// TwinCAT 3 PLC project PLC_1
// ProgramVersion: 3.1.4020.4
// libraries:
//   Tc2_ModbusSrv, * (Beckhoff Automation GmbH)
//   Tc2_Standard, * (Beckhoff Automation GmbH)
//   Tc2_System, * (Beckhoff Automation GmbH)
//   Tc2_TcpIp, * (Beckhoff Automation GmbH)
//   Tc2_Utilities, * (Beckhoff Automation GmbH)
//   Tc3_Module, * (Beckhoff Automation GmbH)
//   VisuDialogs, * (System)
// project tree:
//   DUTs/ E_RobotTaskStates.TcDUT, E_ProcessModes.TcDUT, E_RobotDataRecordingStates.TcDUT, E_UDPConnection.TcDUT, ST_16Bool.TcDUT, ST_Fixture.TcDUT, ST_OptoforceUDPData.TcDUT, ST_OptoforceUDPRequest.TcDUT, ST_Part.TcDUT, ST_RobotTaskStatusInfo.TcDUT, ST_UR.TcDUT
//   DUTs/UR_TCP_IP_Data_Collection_DUTs/ E_RobotTCPReceive.TcDUT, ST_AdditionalInfo.TcDUT, ST_CalibraitonData.TcDUT, ST_CartesianInfo.TcDUT, ST_ConfigurationData.TcDUT, ST_ForceModeData.TcDUT, ST_JointData.TcDUT, ST_KinematicInfo.TcDUT, ST_MasterboardData.TcDUT, ST_PackageInfo.TcDUT, ST_RobotModeData.TcDUT, ST_ToolData.TcDUT
//   / GlobalTextList.TcGTLO, PlcTask.TcTTO, Visualization Manager.TcVMO (not stored)
//   GVLs/ Global.TcGVL, Global_Safety.TcGVL
//   POUs/ FB_CSV_PartDataWriter.TcPOU, FB_CSV_RobotDataWriter.TcPOU, FB_CSV_FTDataWriter.TcPOU, FB_FT_UDPConnection.TcPOU, MAIN.TcPOU, F_Word_To_16Bool.TcPOU, P_InitializeSystem.TcPOU, P_InputOutputHandling.TcPOU, P_Safety.TcPOU, P_TaskHandling.TcPOU
//   POUs/Modbus POUs/ FB_mbReadSingleReg.TcPOU, FB_mbReadRobotTaskStatusInfo.TcPOU, FB_mbWriteRobotTask.TcPOU, FB_mbWriteSingleReg.TcPOU
//   POUs/UR_TCP_IP_Data_Collection/ FB_ParseURData.TcPOU, FB_RobotTCPReceive.TcPOU, F_RecCartesianInfo.TcPOU, F_RecJointData.TcPOU, F_RecRobotModeData.TcPOU, F_RecConfigurationData.TcPOU, F_FindAddr.TcPOU, F_RecForceModeData.TcPOU
//   VISUs/ ForceAndTorque.TcVIS, PositionCheck.TcVIS, Settings.TcVIS, Process.TcVIS, TopVisu.TcVIS
// real-time tasks:
//   TASK PlcTask: cycle T#1ms, priority 20, ADS port 350
// I/O:
//   DEVICE Device 1 (EtherCAT), AmsNetId 5.43.59.116.2.1
//     Term 1 (EK1200) [EK1200-5000 EtherCAT Power supply (2A E-Bus)]
//       SafetyPLC (EL6900) [EL6900, TwinSAFE PLC]
//       Safe In - E-Stop & Reset (EL1904) [EL1904, 4 Ch. Safety Input 24V, TwinSAFE]
//         modules: Module 1 (FSOES)
//       Safe In - Programming Mode (EL1904) [EL1904, 4 Ch. Safety Input 24V, TwinSAFE]
//         modules: Module 1 (FSOES)
//       In - Control Buttons (EL1014) [EL1014 4Ch. Dig. Input 24V, 10µs]
//       In - Unused (EL1014) [EL1014 4Ch. Dig. Input 24V, 10µs]
//       Out - Control Button Ind. (EL2004) [EL2004 4Ch. Dig. Output 24V, 0.5A]
//       Out - Prog. Mode Ind. (EL2004) [EL2004 4Ch. Dig. Output 24V, 0.5A]
//       EtherCAT Extender (EK1110) [EK1110 EtherCAT extension]
//     Term 10 (EK1100) [EK1100 EtherCAT Coupler (2A E-Bus)]
//       In 2/3 wire - Unused 1 (EL1012) [EL1012 2Ch. Dig. Input 24V, 10µs]
//       Safe In - Robot E-Stop Cond. (EL1904) [EL1904, 4 Ch. Safety Input 24V, TwinSAFE]
//         modules: Module 1 (FSOES)
//       Safe In - E-Stop and Mats (EL1904) [EL1904, 4 Ch. Safety Input 24V, TwinSAFE]
//         modules: Module 1 (FSOES)
//       Safe In - Safety Laser A (horizontal) (EL1904) [EL1904, 4 Ch. Safety Input 24V, TwinSAFE]
//         modules: Module 1 (FSOES)
//       Safe In - Safety Laser B (vertical)  (EL1904) [EL1904, 4 Ch. Safety Input 24V, TwinSAFE]
//         modules: Module 1 (FSOES)
//       Safe Out - Robot Safety States (EL2904) [EL2904, 4 Ch. Safety Output 24V, 0.5A, TwinSAFE]
//         modules: Module 1 (FSOES), Module 2 (DO)
//       Out - Stack Lights (EL2008) [EL2008 8Ch. Dig. Output 24V, 0.5A]
//       In - General 1-wire (EL1018) [EL1018 8Ch. Dig. Input 24V, 10µs]
//       In - Unused 3 (EL1114) [EL1114 4Ch. Dig. Input 24V, 10µs, Sensor Power]
//       End Cap (passive) (EL9011) [EL9011 End Terminal]
// variable links:
//   Device 1 (EtherCAT) <-> Device 1 (EtherCAT)/Term 1 (EK1200)/SafetyPLC (EL6900)
//     Term 1 (EK1200)/Safe In - E-Stop & Reset (EL1904)/Module 1 (FSOES)/RxPDO/FSOE <-> ConnectionInputs/Message_3 TxPDO
//     Term 1 (EK1200)/Safe In - E-Stop & Reset (EL1904)/Module 1 (FSOES)/TxPDO/FSOE <-> ConnectionOutputs/Message_3 RxPDO
//     Term 1 (EK1200)/Safe In - Programming Mode (EL1904)/Module 1 (FSOES)/RxPDO/FSOE <-> ConnectionInputs/Message_15 TxPDO
//     Term 1 (EK1200)/Safe In - Programming Mode (EL1904)/Module 1 (FSOES)/TxPDO/FSOE <-> ConnectionOutputs/Message_15 RxPDO
//     Term 10 (EK1100)/Safe In - E-Stop and Mats (EL1904)/Module 1 (FSOES)/RxPDO/FSOE <-> ConnectionInputs/Message_6 TxPDO
//     Term 10 (EK1100)/Safe In - E-Stop and Mats (EL1904)/Module 1 (FSOES)/TxPDO/FSOE <-> ConnectionOutputs/Message_6 RxPDO
//     Term 10 (EK1100)/Safe In - Robot E-Stop Cond. (EL1904)/Module 1 (FSOES)/RxPDO/FSOE <-> ConnectionInputs/Message_14 TxPDO
//     Term 10 (EK1100)/Safe In - Safety Laser A (horizontal) (EL1904)/Module 1 (FSOES)/RxPDO/FSOE <-> ConnectionInputs/Message_16 TxPDO
//     Term 10 (EK1100)/Safe In - Safety Laser A (horizontal) (EL1904)/Module 1 (FSOES)/TxPDO/FSOE <-> ConnectionOutputs/Message_16 RxPDO
//     Term 10 (EK1100)/Safe In - Safety Laser B (vertical)  (EL1904)/Module 1 (FSOES)/RxPDO/FSOE <-> ConnectionInputs/Message_18 TxPDO
//     Term 10 (EK1100)/Safe Out - Robot Safety States (EL2904)/Module 1 (FSOES)/RxPDO/FSOE <-> ConnectionInputs/Message_9 TxPDO
//   Device 1 (EtherCAT) <-> Device 1 (EtherCAT)/Term 10 (EK1100)/Safe In - Robot E-Stop Cond. (EL1904)
//     Term 1 (EK1200)/SafetyPLC (EL6900)/ConnectionOutputs/Message_14 RxPDO <-> Module 1 (FSOES)/TxPDO/FSOE
//   Device 1 (EtherCAT) <-> Device 1 (EtherCAT)/Term 10 (EK1100)/Safe In - Safety Laser B (vertical)  (EL1904)
//     Term 1 (EK1200)/SafetyPLC (EL6900)/ConnectionOutputs/Message_18 RxPDO <-> Module 1 (FSOES)/TxPDO/FSOE
//   Device 1 (EtherCAT) <-> Device 1 (EtherCAT)/Term 10 (EK1100)/Safe Out - Robot Safety States (EL2904)
//     Term 1 (EK1200)/SafetyPLC (EL6900)/ConnectionOutputs/Message_9 RxPDO <-> Module 1 (FSOES)/TxPDO/FSOE
//   PLC_1/PLC_1 Instance <-> Device 1 (EtherCAT)/Term 1 (EK1200)/In - Control Buttons (EL1014)
//     PlcTask Inputs/Global.pbStart <-> Channel 1/Input
//     PlcTask Inputs/Global.pbStop <-> Channel 2/Input
//   PLC_1/PLC_1 Instance <-> Device 1 (EtherCAT)/Term 1 (EK1200)/Out - Control Button Ind. (EL2004)
//     PlcTask Outputs/Global.indStartPB <-> Channel 3/Output
//     PlcTask Outputs/Global.indStopPB <-> Channel 4/Output
//     PlcTask Outputs/Global_Safety.CPEStopIND <-> Channel 1/Output
//     PlcTask Outputs/Global_Safety.CPFaultIND <-> Channel 2/Output
//   PLC_1/PLC_1 Instance <-> Device 1 (EtherCAT)/Term 1 (EK1200)/Out - Prog. Mode Ind. (EL2004)
//     PlcTask Outputs/Global_Safety.CPEProgramModeIND <-> Channel 1/Output
//   PLC_1/PLC_1 Instance <-> Device 1 (EtherCAT)/Term 1 (EK1200)/Safe In - E-Stop & Reset (EL1904)
//     PlcTask Inputs/Global_Safety.ResetPB <-> Module 1 (FSOES)/TxPDO/FSOE/InputChannel3
//   PLC_1/PLC_1 Instance <-> Device 1 (EtherCAT)/Term 1 (EK1200)/SafetyPLC (EL6900)
//     PlcTask Inputs/Global_Safety.NotInEStop <-> StandardInputs/Standard Out Var 22
//     PlcTask Inputs/Global_Safety.NotInRedSpeed <-> StandardInputs/Standard Out Var 20
//     PlcTask Inputs/Global_Safety.NotInSafeStop <-> StandardInputs/Standard Out Var 21
//     PlcTask Inputs/Global_Safety.ProgramModeActive <-> StandardInputs/Standard Out Var 25
//     PlcTask Inputs/Global_Safety.SafetyPLCState <-> TwinSAFE Group Info Data/TwinSafeGroup1 Info Data/State
//     PlcTask Outputs/Global_Safety.ErrorAck <-> StandardOutputs/Standard In Var 11
//   PLC_1/PLC_1 Instance <-> Device 1 (EtherCAT)/Term 10 (EK1100)/In - General 1-wire (EL1018)
//     PlcTask Inputs/Global.bPosSensorState <-> Channel 1/Input
//   PLC_1/PLC_1 Instance <-> Device 1 (EtherCAT)/Term 10 (EK1100)/Out - Stack Lights (EL2008)
//     PlcTask Outputs/Global_Safety.UR3AmberIND <-> Channel 7/Output
//     PlcTask Outputs/Global_Safety.UR5AmberIND <-> Channel 3/Output
//     PlcTask Outputs/Global_Safety.UR3BlueIND <-> Channel 5/Output
//     PlcTask Outputs/Global_Safety.UR5BlueIND <-> Channel 1/Output
//     PlcTask Outputs/Global_Safety.UR3GreenIND <-> Channel 6/Output
//     PlcTask Outputs/Global_Safety.UR5GreenIND <-> Channel 2/Output
//     PlcTask Outputs/Global_Safety.UR3RedIND <-> Channel 8/Output
//     PlcTask Outputs/Global_Safety.UR5RedIND <-> Channel 4/Output

CONFIGURATION PLC_1
    RESOURCE PLC ON TwinCAT3
        TASK PlcTask(INTERVAL := T#1ms, PRIORITY := 20);
        PROGRAM MAIN WITH PlcTask : MAIN;
    END_RESOURCE
END_CONFIGURATION

// ---- DUTs/E_RobotTaskStates.TcDUT
{attribute 'qualified_only'}
{attribute 'strict'}
TYPE E_RobotTaskStates :
(
	Idle,
	TaskTypeSelection,
	TaskSelection,
	TaskAssignment,
	TaskAssignment_Wait,
	TaskExecution
);
END_TYPE

// ---- DUTs/E_ProcessModes.TcDUT
{attribute 'qualified_only'}
{attribute 'strict'}
TYPE E_ProcessModes :
(
	Idle,
	Running,
	Stopping
);
END_TYPE

// ---- DUTs/E_RobotDataRecordingStates.TcDUT
{attribute 'qualified_only'}
{attribute 'strict'}
TYPE E_RobotDataRecordingStates :
(
	Idle,
	CollectData,
	CollectData_Wait,
	RecordData,
	RecordData_Wait,
	HandleError
);
END_TYPE

// ---- DUTs/E_UDPConnection.TcDUT
{attribute 'qualified_only'}
{attribute 'strict'}
TYPE E_UDPConnection :
(
	Idle,
	Connect_Start,
	Connect_Wait,
	Request_Start,
	Request_Wait,
	Receive_Start,
	Receive_Wait,
	RecordData,
	Close_Start,
	Close_Wait,
	HandleError
);
END_TYPE

// ---- DUTs/ST_16Bool.TcDUT
TYPE ST_16Bool :
STRUCT
	var1 : BOOL;
	var2 : BOOL;
	var3 : BOOL;
	var4 : BOOL;
	var5 : BOOL;
	var6 : BOOL;
	var7 : BOOL;
	var8 : BOOL;
	var9 : BOOL;
	var10 : BOOL;
	var11 : BOOL;
	var12 : BOOL;
	var13 : BOOL;
	var14 : BOOL;
	var15 : BOOL;
	var16 : BOOL;

END_STRUCT
END_TYPE

// ---- DUTs/ST_Fixture.TcDUT
TYPE ST_Fixture :
STRUCT
	// Fixture Constants
	nWorkframe : WORD;
	
	// Fixture State
	bReserved : BOOL;
	
	// Part
	stPart : ST_Part := (bExists := FALSE, bComplete := FALSE);
	
END_STRUCT
END_TYPE

// ---- DUTs/ST_OptoforceUDPData.TcDUT
TYPE ST_OptoforceUDPData :
STRUCT
	HS_sequence : UDINT; // The sequence number of the current HS UDP record
	FT_sequence : UDINT; // The internal sample counter of the DAQ
	Status : UDINT; // Status word of the sensor and DAQ
	Fx : DINT; // X-axis force in 32 bit Counts*
	Fy : DINT; // Y-axis force in 32 bit Counts*
	Fz : DINT; // Z-axis force in 32 bit Counts*
	Tx : DINT; // X-axis torque in 32 bit Counts* (0 if not available)
	Ty : DINT; // Y-axis torque in 32 bit Counts* (0 if not available)
	Tz : DINT; // Z-axis torque in 32 bit Counts* (0 if not available)
END_STRUCT
END_TYPE

// ---- DUTs/ST_OptoforceUDPRequest.TcDUT
TYPE ST_OptoforceUDPRequest :
STRUCT
	Header : UINT; // Must be 0x1234
	Command : UINT; // Value according to the command table
	Data : UDINT; // data according to the actual command
END_STRUCT
END_TYPE

// ---- DUTs/ST_Part.TcDUT
TYPE ST_Part :
STRUCT
	// Part State
	bExists : BOOL;
	bComplete : BOOL;
	
	// Part Attributes
	nPartType : WORD;
	
	// Process Time
	rtUR3TimePartAdded : LWORD;
	rtUR5TimePartAdded : LWORD;
	ntPartAdded : ULINT;
	
	// Pick and Place from Input to WF
	ntPickFromInputAssigned : ULINT;
	ntInputPartPicked : ULINT;
	ntInputPartPlaced : ULINT;
	ntPlaceInWFComplete : ULINT;
	
	// Task on Part
	ntTaskAssigned : ULINT;
	ntTaskActionStart : ULINT;
	ntTaskActionComplete : ULINT;
	ntTaskComplete : ULINT;
	
	// Pick and Place from WF to Output
	ntPickFromWFAssigned : ULINT;
	ntOutputPartPicked : ULINT;
	ntOutputPartPlaced : ULINT;
	ntPlaceInOutputComplete : ULINT;
	
	// Part removed from cell
	ntPartRemoved : ULINT;
	
	// Process Record Data
	ntTimeInWorkfixture : REAL;
	nWorkFixture : WORD;
	nInputPosition : WORD;
	nOutputPosition : WORD;
	nPartNumber : WORD;
	
	
END_STRUCT
END_TYPE

// ---- DUTs/ST_RobotTaskStatusInfo.TcDUT
TYPE ST_RobotTaskStatusInfo :
STRUCT
	nRobotTaskStatus : WORD;
	nZoneOccupied : WORD;
	bInTask : BOOL;
	bPerformingTaskAction : BOOL;
	sRobotStatus : STRING;

END_STRUCT
END_TYPE

// ---- DUTs/ST_UR.TcDUT
TYPE ST_UR :
STRUCT
	// Robot Setup Variables (Constants)
	IP: STRING(15);
	mbPort: UINT := 502;
	unitID: BYTE := 255;

	// MODBUS Robot Data 
	mode : WORD;
	
	// TCP/IP Connection Data
	RobotModeData : ST_RobotModeData;
	JointData : ST_JointData;
	ConfigurationData : ST_ConfigurationData;
	CartesianInfo : ST_CartesianInfo;
	ForceModeData : ST_ForceModeData;
	
	// Induced Joint Error 
	InducedJErrorType : WORD; // 0 none, 1 slip, 2 backlash
	InducedJointError : ARRAY [1..6] OF WORD;
	
END_STRUCT
END_TYPE

// ---- DUTs/UR_TCP_IP_Data_Collection_DUTs/E_RobotTCPReceive.TcDUT
{attribute 'qualified_only'}
{attribute 'strict'}
TYPE E_RobotTCPReceive :
(
	Idle,
	Connect_Start,
	Connect_Wait,
	Receive_Start,
	Receive_Wait,
	ParseData,
	RecordData,
	RecordData_Wait,
	Close_Start,
	Close_Wait,
	HandleError
);
END_TYPE

// ---- DUTs/UR_TCP_IP_Data_Collection_DUTs/ST_AdditionalInfo.TcDUT
TYPE ST_AdditionalInfo :
STRUCT
	// Additional Info (Value 8)
	AdditionalInfo: ARRAY [1..8] OF BYTE;

END_STRUCT
END_TYPE

// ---- DUTs/UR_TCP_IP_Data_Collection_DUTs/ST_CalibraitonData.TcDUT
TYPE ST_CalibraitonData :
STRUCT
	// Calibration Data (Value 9)
	CalibrationData: ARRAY [1..53] OF BYTE;		
END_STRUCT
END_TYPE

// ---- DUTs/UR_TCP_IP_Data_Collection_DUTs/ST_CartesianInfo.TcDUT
TYPE ST_CartesianInfo :
STRUCT
	// Cartesian Info (Value 4)
	// CartesianInfo: ARRAY [1..101] OF BYTE;
	PackageLength: UDINT;
	PackageType: USINT;
	ToolX: LREAL;
	ToolY: LREAL;
	ToolZ: LREAL;
	ToolRx: LREAL;
	ToolRy: LREAL;
	ToolRz: LREAL;
	TCPOffsetX: LREAL;
	TCPOffsetY: LREAL;
	TCPOffsetZ: LREAL;
	TCPOffsetRx: LREAL;
	TCPOffsetRy: LREAL;
	TCPOffsetRz: LREAL;
	
	arrVarLength: ARRAY [1..14] OF USINT := [4,1,12(8)];
END_STRUCT
END_TYPE

// ---- DUTs/UR_TCP_IP_Data_Collection_DUTs/ST_ConfigurationData.TcDUT
TYPE ST_ConfigurationData :
STRUCT
	// Configuration Data (Value 6)
	PackageLength: UDINT;
	PackageType: USINT;		
	// Joint min and max position, speed and accel
		JointMinMax: ARRAY [1..192] OF BYTE;		
	// Default TCP and Tool speed and accel limits	
		ToolLimits: ARRAY [1..32] OF BYTE;
	// Other tool info	
		EqRadius: LREAL;
	// DH Parameters
		DHa: ARRAY [1..6] OF LREAL;	
		DHd: ARRAY [1..6] OF LREAL;							
		DHalpha: ARRAY [1..6] OF LREAL;							
		DHtheta: ARRAY [1..6] OF LREAL;				
	// Other Robot info			
		OtherConfigData: ARRAY [1..16] OF BYTE;		
		
arrVarLength: ARRAY [1..59] OF USINT := [4,1,6(8),6(8),6(8),6(8),5(8),6(8),6(8),6(8),6(8),4(4)];
END_STRUCT
END_TYPE

// ---- DUTs/UR_TCP_IP_Data_Collection_DUTs/ST_ForceModeData.TcDUT
TYPE ST_ForceModeData :
STRUCT
	// Force Mode Data (Value 7)
	//ForceModeData: ARRAY [1..61] OF BYTE;
	PackageLength: UDINT;
	PackageType: USINT;
	FmodeX: LWORD;
	FmodeY: LWORD;
	FmodeZ: LWORD;
	FmodeRx: LWORD;
	FmodeRy: LWORD;
	FmodeRz: LWORD;
	TCPDexterity: LWORD;
	
	arrVarLength: ARRAY [1..9] OF USINT := [4,1,7(8)];

END_STRUCT
END_TYPE

// ---- DUTs/UR_TCP_IP_Data_Collection_DUTs/ST_JointData.TcDUT
TYPE ST_JointData :
STRUCT
	// Joint Data (Value 1)
	PackageLength: UDINT;
	PackageType: USINT;
	// Joint 1		
		j1_qactual: LREAL;
		j1_qtarget: LREAL;			
		j1_qdactual: LREAL;			
		j1_Iactual: REAL;		
		j1_Vactual: REAL;			
		j1_Tmotor: REAL;			
		j1_Tmicro: REAL;	// Dont use obsolete
		j1_JointMode: USINT; 
	// Joint 2
		j2_qactual: LREAL;
		j2_qtarget: LREAL;			
		j2_qdactual: LREAL;			
		j2_Iactual: REAL;		
		j2_Vactual: REAL;			
		j2_Tmotor: REAL;			
		j2_Tmicro: REAL;	// Dont use obsolete
		j2_JointMode: USINT; 
	// Joint 3
		j3_qactual: LREAL;
		j3_qtarget: LREAL;			
		j3_qdactual: LREAL;			
		j3_Iactual: REAL;		
		j3_Vactual: REAL;			
		j3_Tmotor: REAL;			
		j3_Tmicro: REAL;	// Dont use obsolete
		j3_JointMode: USINT; 
	// Joint 4
		j4_qactual: LREAL;
		j4_qtarget: LREAL;			
		j4_qdactual: LREAL;			
		j4_Iactual: REAL;		
		j4_Vactual: REAL;			
		j4_Tmotor: REAL;			
		j4_Tmicro: REAL;	// Dont use obsolete
		j4_JointMode: USINT; 
	// Joint 5
		j5_qactual: LREAL;
		j5_qtarget: LREAL;			
		j5_qdactual: LREAL;			
		j5_Iactual: REAL;		
		j5_Vactual: REAL;			
		j5_Tmotor: REAL;			
		j5_Tmicro: REAL;	// Dont use obsolete
		j5_JointMode: USINT; 
	// Joint 6
		j6_qactual: LREAL;
		j6_qtarget: LREAL;			
		j6_qdactual: LREAL;			
		j6_Iactual: REAL;		
		j6_Vactual: REAL;			
		j6_Tmotor: REAL;			
		j6_Tmicro: REAL;	// Dont use obsolete
		j6_JointMode: USINT; 
	
	// Packet Item Length Info
	arrVarLength: ARRAY [1..53] OF USINT := [4,1,3(8),4(4),1,3(8),4(4),1,3(8),4(4),1,3(8),4(4),1,3(8),4(4),1,3(8),4(4),1];
END_STRUCT
END_TYPE

// ---- DUTs/UR_TCP_IP_Data_Collection_DUTs/ST_KinematicInfo.TcDUT
TYPE ST_KinematicInfo :
STRUCT
	// Kinematic Info (Value 5)
	KinematicInfo: ARRAY [1..225] OF BYTE;

END_STRUCT
END_TYPE

// ---- DUTs/UR_TCP_IP_Data_Collection_DUTs/ST_MasterboardData.TcDUT
TYPE ST_MasterboardData :
STRUCT
	// Masterboard Data (Value 3)
	MasterboardData: ARRAY [1..74] OF BYTE;

END_STRUCT
END_TYPE

// ---- DUTs/UR_TCP_IP_Data_Collection_DUTs/ST_PackageInfo.TcDUT
TYPE ST_PackageInfo :
STRUCT
	PackageLength: UDINT;
	MessageType: USINT;
END_STRUCT
END_TYPE

// ---- DUTs/UR_TCP_IP_Data_Collection_DUTs/ST_RobotModeData.TcDUT
TYPE ST_RobotModeData :
STRUCT
	(* Robot Mode Data (Value 0) Length: 46 Bytes *)
	PackageLength: UDINT;
	PackageType: USINT;
	Timestamp: LWORD;
	PhysicalRobotConnected: BYTE; 
	RealRobotEnabled: BYTE; 
	RobotPowerOn: BYTE; 
	EmergencyStopped: BYTE;
	ProtectiveStopped: BYTE;
	ProgramRunning: BYTE;
	ProgramPaused: BYTE;
	RobotMode: USINT;
	ControlMode: USINT;
	TargetSpeedFraction: LWORD;
	SpeedScaling: LWORD;
	TargetSpeedFractionLimit: LWORD;
	
	arrVarLength: ARRAY [1..15] OF USINT := [4,1,8,9(1),3(8)];
	
END_STRUCT
END_TYPE

// ---- DUTs/UR_TCP_IP_Data_Collection_DUTs/ST_ToolData.TcDUT
TYPE ST_ToolData :
STRUCT
	// Tool Data (Value 2)
	ToolData: ARRAY [1..37] OF BYTE;
END_STRUCT
END_TYPE

// ---- GVLs/Global.TcGVL
{attribute 'qualified_only'}
VAR_GLOBAL
	(* Robot Data *)
	
	// Robot Structures
	stUR5 : ST_UR := (IP := '192.168.1.5'); // UR5
	stUR3 : ST_UR := (IP := '192.168.1.3'); // UR3
	bUR5NewTCPData : BOOL;
	bUR3NewTCPData : BOOL;
	
	bUR3InTask : BOOL;
	bUR5InTask : BOOL;
	
	
	// Universal Robot MODBUS Addresses (16 bit registers)
	ModeAddr: WORD := 258; // Robot Mode MODBUS Address
	
	
	(* Workcell Variables *)
	
	// Process Control
	bActivatePartDataRecording : BOOL;
	bActivateTaskAssignment : BOOL;
	bActivateTCPIPDataCollection : BOOL;
	bActivateTCPIPDataRecording : BOOL;
	bActivateFTDataCollection : BOOL;
	bActivateFTDataRecording : BOOL;
	
	// Drawing Task control variable (Togled on setting visualization)
	// Box and Circle is Task 0 (1 in URScript) and NIST Draw is Task 1 (2 in URScript)
	nActiveUR3Task : WORD; // 0 Box and Circle, 1 NIST Logo, 2 Reserved
	
	// ADS Control Variables
	bCycleStart : BOOL;
	bCycleStop : BOOL;
	bResetPartCount : BOOL;
	
	// Fixtures
	bPosSensorReserved: BOOL;
	nNumWorkFixtures : INT := 2;
	arrWorkFixtures : ARRAY [0..2] OF ST_Fixture := [
									(nWorkframe := 0),
									(nWorkframe := 1), 
									(nWorkframe := 2)];
	nNumInputFixtures : INT := 1; // 1 fixture for setup 1 can be made multiple for trays/batch
	arrInputFixtures : ARRAY [0..4] OF ST_Fixture:= [
									(nWorkframe := 0),
									(nWorkframe := 1), 
									(nWorkframe := 2),
									(nWorkframe := 3), 
									(nWorkframe := 4)];
	nNumOutputFixtures : INT := 1; // 1 fixture for setup 1 can be made multiple for trays/batch
	arrOutputFixtures : ARRAY [0..4] OF ST_Fixture:= [
									(nWorkframe := 0),
									(nWorkframe := 1), 
									(nWorkframe := 2),
									(nWorkframe := 3), 
									(nWorkframe := 4)];
									
	
	// Parts
	stNullPart : ST_Part;
	stPartInTransit : ST_Part;
	
	// Time
	nCurrentTime : ULINT; // Current windows time
	nStartTime : ULINT;
	
	// I/O on EtherCAT
	pbStart AT %I*: BOOL; 		// Start Button on Control Pendant (NO)
	pbStop AT %I*: BOOL;		// Stop Button on Control Pendant (NC)
	
	indStartPB AT %Q*: BOOL;
	indStopPB AT %Q*: BOOL;
	
	
	(* HMI Variables for Display *)
	// Unused
	
	(* History *)
	CompletedParts : ARRAY [1..10] OF ST_Part;
	nPartsStarted : WORD;
	nPartsCompleted : ULINT;
	nTotalPartTime : ULINT;
	nAveragePartTime : LREAL;
	
	
	(* Health Data *)
	bPosSensorState AT %I* : BOOL; // Position Sensor
	bEnablePosCheck : BOOL;
	bForcePosCheck : BOOL;
	nPartsSincePosCheck : UINT;
	nPosCheckThreshold : UINT := 100;
	
	UR3PosCheck : ARRAY [1..2] OF BOOL; // ST_16Bool for UR integrated sensor
	UR5PosCheck : ARRAY [1..5] OF BOOL; // ST_16Bool for UR integrated sensor
	
	(* Other *)
	stFTData : ST_OptoforceUDPData;
	
	
	
END_VAR

// ---- GVLs/Global_Safety.TcGVL
{attribute 'qualified_only'}
VAR_GLOBAL
	// Safety Related Variables (Excluding Data from Robot)
	
	// Safety Inputs
	ResetPB AT %I*: BOOL;
	NotInRedSpeed AT %I*: BOOL;
	NotInSafeStop AT %I*: BOOL;
	NotInEStop AT %I*: BOOL;
	ProgramModeActive AT %I*: BOOL;
	
	SafetyPLCState AT %I*: USINT;
	
	// Safety Outputs
	ErrorAck AT %Q*: BOOL;
	
	// Stack Lights
	UR3RedIND AT %Q*: BOOL;
	UR3AmberIND AT %Q*: BOOL;
	UR3GreenIND AT %Q*: BOOL;
	UR3BlueIND AT %Q*: BOOL;
	UR5RedIND AT %Q*: BOOL;
	UR5AmberIND AT %Q*: BOOL;
	UR5GreenIND AT %Q*: BOOL;
	UR5BlueIND AT %Q*: BOOL;
	
	// Control Pendant Indicators
	CPEStopIND AT %Q*: BOOL;
	CPFaultIND AT %Q*: BOOL;
	CPEProgramModeIND AT %Q*: BOOL;
END_VAR

// ---- POUs/MAIN.TcPOU
PROGRAM MAIN
VAR
	// Data Recording
	fbUR5tcp : FB_RobotTCPReceive := (Robot := 'UR5');
	fbUR3tcp : FB_RobotTCPReceive := (Robot := 'UR3');
	eRobotDataRecordingState : E_RobotDataRecordingStates;
	
	
	// Optoforce
	fbRecFTData : FB_FT_UDPConnection;

	
	// Triggers
	StartTrig: R_TRIG;
	StopTrig: F_TRIG;
	
	// Procees State Machine
	eProcessMode : E_ProcessModes;
	sProcessState : STRING;
	

	
END_VAR

(* =======================================================
Update veriables on every cycle
======================================================= *)
// Record time every cycle
Global.nCurrentTime := F_GetSystemTime();

// Triggers for start and stop buttons on control pendant
StartTrig(CLK := Global.pbStart); // Start
StopTrig(CLK := Global.pbStop); // Stop

(* =======================================================
Process Mode State Machine 
======================================================= *)
// Interrupts
	// Stop Button
	IF StopTrig.Q OR Global.bCycleStop THEN 
		eProcessMode := E_ProcessModes.Stopping;
		Global.bCycleStop := FALSE;
	END_IF
// State Machine
CASE eProcessMode OF
	E_ProcessModes.Idle:
		sProcessState := 'Idle';
		// Wait for start button to trigger
		IF StartTrig.Q OR Global.bCycleStart THEN
			eProcessMode := E_ProcessModes.Running;
			Global.bCycleStart := FALSE;
		END_IF
		Global.indStartPB := FALSE;
		Global.indStopPB := TRUE;
		
	E_ProcessModes.Running:
		sProcessState := 'Assigning Tasks';
		Global.bActivateTaskAssignment := TRUE;
		Global.indStartPB := TRUE;
		Global.indStopPB := FALSE;
	E_ProcessModes.Stopping:
		sProcessState := 'Performing Last Tasks';
		Global.bActivateTaskAssignment := FALSE;
		eProcessMode := E_ProcessModes.Idle;
END_CASE

(* =======================================================
Data Collection Processes
======================================================= *)


// Enable TCP/IP Data collection from robots
fbUR5tcp.bEnable := Global.bActivateTCPIPDataCollection;
fbUR3tcp.bEnable := Global.bActivateTCPIPDataCollection;
IF Global.bActivateTCPIPDataCollection THEN
	fbUR5tcp.bRecordData := Global.bActivateTCPIPDataRecording;
	fbUR3tcp.bRecordData := Global.bActivateTCPIPDataRecording;
ELSE
	fbUR5tcp.bRecordData := FALSE;
	fbUR3tcp.bRecordData := FALSE;
END_IF


// Enable UDP Data collection from Force and Torque Sensor
fbRecFTData.bEnable := Global.bActivateFTDataCollection;
IF Global.bActivateFTDataCollection THEN
	fbRecFTData.bRecordData := Global.bActivateFTDataRecording;
ELSE
	fbRecFTData.bRecordData := FALSE;
END_IF

(* =======================================================
Function block Calls
======================================================= *)
fbUR5tcp();
fbUR3tcp();
fbRecFTData(stOptoforceData => Global.stFTData );

(* =======================================================
Sub-programs that run all the time
======================================================= *)
P_Safety(); // Handle Safety Funftions and collects safety related data
P_InputOutputHandling();
P_TaskHandling();

(* =======================================================
Automated Experiment Data Cleaning / Reset
======================================================= *)
IF Global.bResetPartCount THEN
	Global.nPartsStarted := 0;
	Global.nPartsCompleted := 0;
	Global.nTotalPartTime := 0;
	Global.nAveragePartTime := 0;
	Global.bResetPartCount := FALSE;
END_IF

END_PROGRAM

// ---- POUs/UR_TCP_IP_Data_Collection/FB_RobotTCPReceive.TcPOU
FUNCTION_BLOCK FB_RobotTCPReceive
VAR_INPUT
	bEnable : BOOL;
	Robot : STRING;
	bRecordData : BOOL;

END_VAR
VAR_OUTPUT
	bBusy : BOOL;
	bConnected : BOOL;
	bError : BOOL;
	
	
END_VAR
VAR
	data : ARRAY [1..1500] OF BYTE;
	packageData : ARRAY [1..500] OF BYTE;
	eState : E_RobotTCPReceive;
	
	fbSocketConnect : FB_SocketConnect := (sSrvNetId := '', tTimeout := DEFAULT_ADS_TIMEOUT);
	fbSocketClose : FB_SocketClose := (sSrvNetId := '', tTimeout := DEFAULT_ADS_TIMEOUT);
	fbSocketReceive : FB_SocketReceive := (sSrvNetId := '', tTimeout := DEFAULT_ADS_TIMEOUT, cbLen := 1500); //1076
	fbParseURData : FB_ParseURData;
	fbRecordData : FB_CSV_RobotDataWriter;
	
	hSocket1: T_HSOCKET;
	bParsingData: BOOL;

END_VAR

// TCP/IP Messaging Case
CASE eState OF
	
	E_RobotTCPReceive.Idle:
		IF bEnable THEN
			bBusy := TRUE;
			IF NOT bConnected THEN
				eState := E_RobotTCPReceive.Connect_Start;
			ELSE
				eState := E_RobotTCPReceive.Receive_Start;
			END_IF
		ELSIF bConnected THEN
			eState := E_RobotTCPReceive.Close_Start;
		END_IF
	
	E_RobotTCPReceive.Connect_Start:
		fbSocketConnect.bExecute := TRUE;
		fbSocketConnect.nRemotePort := 30001;
		IF Robot='UR3' THEN
			fbSocketConnect.sRemoteHost := Global.stUR3.IP;	
		ELSIF Robot='UR5' THEN
			fbSocketConnect.sRemoteHost := Global.stUR5.IP;
		ELSE
			eState := E_RobotTCPReceive.HandleError;
		END_IF
		eState := E_RobotTCPReceive.Connect_Wait;
		
	E_RobotTCPReceive.Connect_Wait:
		fbSocketConnect.bExecute := FALSE;	
		IF fbSocketConnect.bError THEN
			eState := E_RobotTCPReceive.HandleError;
		ELSIF NOT fbSocketConnect.bBusy THEN
			bConnected := TRUE;
			hSocket1 := fbSocketConnect.hSocket;
			eState := E_RobotTCPReceive.Idle;
		END_IF
		
	E_RobotTCPReceive.Receive_Start:
		fbSocketReceive.bExecute := TRUE;
		fbSocketReceive.hSocket := hSocket1;
		fbSocketReceive.pDest := ADR(data);
		eState := E_RobotTCPReceive.Receive_Wait;
	
	E_RobotTCPReceive.Receive_Wait:
		fbSocketReceive.bExecute := FALSE;
		IF fbSocketReceive.bError THEN
			eState := E_RobotTCPReceive.HandleError;
		ELSIF NOT fbSocketReceive.bBusy THEN
			bParsingData := TRUE;
			eState := E_RobotTCPReceive.ParseData;
		END_IF
		
	E_RobotTCPReceive.ParseData:
		IF bParsingData THEN	
			fbParseURData( data := data, Robot:=Robot);  // Parse and Record UR Data
			bParsingData := FALSE;
			//eState := E_RobotTCPReceive.Idle;
		ELSE
			eState := E_RobotTCPReceive.Idle;
		END_IF
		IF bRecordData THEN
			fbRecordData.bEnable := TRUE;
			IF Robot='UR3' THEN
				fbRecordData.sFileName := 'UR3Data';
				fbRecordData.stRobotData := Global.stUR3;
			ELSIF Robot='UR5' THEN
				fbRecordData.sFileName := 'UR5Data';
				fbRecordData.stRobotData := Global.stUR5;
			END_IF

			fbRecordData.bWriteLine := TRUE;
			
			eState := E_RobotTCPReceive.RecordData_Wait;
		ELSE 
			eState := E_RobotTCPReceive.Idle;
			fbRecordData.bEnable := FALSE;
		END_IF
		
	E_RobotTCPReceive.RecordData_Wait:
		IF fbRecordData.bError THEN
			eState := E_RobotTCPReceive.HandleError;
		ELSIF NOT fbRecordData.bBusy THEN
			eState := E_RobotTCPReceive.Idle;
		END_IF
		
	E_RobotTCPReceive.Close_Start:
		fbSocketClose.bExecute := TRUE;
		fbSocketClose.hSocket := hSocket1;
		eState := E_RobotTCPReceive.Close_Wait;
	
	E_RobotTCPReceive.Close_Wait:
		fbSocketClose.bExecute := FALSE;
		IF fbSocketClose.bError THEN
				eState := E_RobotTCPReceive.HandleError;
		ELSIF NOT fbSocketClose.bBusy THEN
			bConnected := FALSE;
			MEMSET(ADR(hSocket1),0,SIZEOF(hSocket1));
			bBusy := FALSE;
			bError := FALSE;
			eState := E_RobotTCPReceive.Idle;
		END_IF
		
	E_RobotTCPReceive.HandleError:
		bError := TRUE;
		IF bConnected THEN
			eState := E_RobotTCPReceive.Close_Start;
		ELSE
			bBusy := FALSE;
			eState := E_RobotTCPReceive.Idle;
		END_IF
		
END_CASE

fbRecordData();
fbSocketConnect();
fbSocketReceive();
fbSocketClose();

END_FUNCTION_BLOCK

// ---- POUs/UR_TCP_IP_Data_Collection/FB_ParseURData.TcPOU
FUNCTION_BLOCK FB_ParseURData
VAR_INPUT
	Robot: STRING;
	data: ARRAY [1..1500] OF BYTE;
END_VAR
VAR_OUTPUT

END_VAR
VAR
	stMessageData: ST_PackageInfo;
	nMessageLength: UDINT;
	nPackageLength: UDINT;
	nMessageType: USINT;
	nPackageType: USINT;
	
	nNextStart: UDINT;
	nRecordIndex: INT;
	arrPackageData: ARRAY [1..500] OF BYTE;
END_VAR

(* Find Total Message Length and Type *)
MEMMOVE(ADR(stMessageData),ADR(data[1]),5);
nMessageLength := BE32_TO_HOST(stMessageData.PackageLength);			// Length of message from Robot
nMessageType := stMessageData.MessageType;								// Type of message from robot 
nNextStart := 6;														// Next byte index in data that is relevant

(* Handle Message Type 16 (Robot State) *)
IF nMessageType=16 THEN
	FOR nRecordIndex := 1 TO 11 DO										// For each of the possible sub-package types (11 possible)
		(* Extract next sub-package length and type *)
		MEMMOVE(ADR(stMessageData),ADR(data[nNextStart]),5);			// Move package length and type to interpretable structure 
		nPackageLength := BE32_TO_HOST(stMessageData.PackageLength);	// Package Length (with conversion)
		nPackageType := stMessageData.MessageType;						// Package type
		MEMMOVE(ADR(arrPackageData),ADR(data[nNextStart]),nPackageLength);	// Move entire package to a buffer array
		(* Extract Data to structure according to data package type *)
		IF nPackageType=0 THEN											// If package type zero
			IF Robot='UR5' THEN
				// Call function to mode data from the buffer to the predefined structure
				Global.stUR5.RobotModeData := F_RecRobotModeData(arrPackageData);
			ELSIF Robot='UR3' THEN
				Global.stUR3.RobotModeData := F_RecRobotModeData(arrPackageData);
			END_IF
			
		ELSIF nPackageType=1 THEN
			IF Robot='UR5' THEN
				Global.stUR5.JointData := F_RecJointData(arrPackageData);
			ELSIF Robot='UR3' THEN
				Global.stUR3.JointData := F_RecJointData(arrPackageData);
			END_IF
		ELSIF nPackageType=4 THEN
			IF Robot='UR5' THEN
				Global.stUR5.CartesianInfo := F_RecCartesianInfo(arrPackageData);
			ELSIF Robot='UR3' THEN
				Global.stUR3.CartesianInfo := F_RecCartesianInfo(arrPackageData);
			END_IF			
		ELSIF nPackageType=6 THEN
			IF Robot='UR5' THEN
				Global.stUR5.ConfigurationData := F_RecConfigurationData(arrPackageData);
			ELSIF Robot='UR3' THEN
				Global.stUR3.ConfigurationData := F_RecConfigurationData(arrPackageData);
			END_IF
		ELSIF nPackageType=7 THEN
			IF Robot='UR5' THEN
				Global.stUR5.ForceModeData := F_RecForceModeData(arrPackageData);
			ELSIF Robot='UR3' THEN
				Global.stUR3.ForceModeData := F_RecForceModeData(arrPackageData);
			END_IF
		END_IF
		nNextStart := nNextStart + nPackageLength; // Increment next index of interest in data
		IF nNextStart>nMessageLength THEN // Exit for loop if all data has been parsed
			EXIT;
		END_IF
	END_FOR
END_IF

END_FUNCTION_BLOCK

// ---- POUs/UR_TCP_IP_Data_Collection/F_RecRobotModeData.TcPOU
FUNCTION F_RecRobotModeData : ST_RobotModeData								// Different for different structures
VAR_INPUT
	data: ARRAY [1..500] OF BYTE;
END_VAR
VAR
	nNumOfVar: UINT;
	nIndex: UINT;
	pAddrTo: POINTER TO ST_RobotModeData;
	nAddrTo: POINTER TO ST_RobotModeData;
	PAddrFrom: POINTER TO ARRAY [1..500] OF BYTE;
	nByteCount: UINT;
	
	n2Byte : UINT;
	n4Byte : UDINT;
	n8Byte : ULINT;
	adr2Byte: POINTER TO UINT;
	adr4Byte: POINTER TO UDINT;
	adr8Byte: POINTER TO ULINT;
	nCurrentVarLength: USINT;
END_VAR

nNumOfVar := SIZEOF(F_RecRobotModeData.arrVarLength);						// Different for different structures
pAddrTo := ADR(F_RecRobotModeData);											// Different for different structures
PAddrFrom := ADR(data);
adr2Byte := ADR(n2Byte);
adr4Byte := ADR(n4Byte);
adr8Byte := ADR(n8Byte);

FOR nIndex := 1 TO nNumOfVar DO
	nCurrentVarLength := F_RecRobotModeData.arrVarLength[nIndex];			// Different for different structures
	
	(* Determine byte address to save item to *)
	nByteCount := nByteCount + nCurrentVarLength;
	IF nByteCount=8 THEN
		pAddrTo := pAddrTo;
		nByteCount := 0;
	ELSIF nByteCount>8 THEN
		pAddrTo := pAddrTo + 16 - nByteCount;
		nByteCount := 0;
	ELSE
		pAddrTo := pAddrTo;
	END_IF
	nAddrTo := F_FindAddr(pAddrTo,nByteCount);
	
	(* Convert Data based on size of item (in bytes) *)
	IF nCurrentVarLength=8 THEN
		MEMCPY(adr8Byte, pAddrFrom, 8);
		n8Byte := BE64_TO_HOSTEX(n8Byte);
		MEMCPY(pAddrTo, adr8Byte, 8);
	ELSIF nCurrentVarLength=4 THEN
		MEMCPY(adr4Byte, pAddrFrom, 8);
		n4Byte := BE32_TO_HOST(n4Byte);
		MEMCPY(pAddrTo, adr4Byte, 8);
	ELSIF nCurrentVarLength=2 THEN
		MEMCPY(adr2Byte, pAddrFrom, 8);
		n2Byte := BE16_TO_HOST(n2Byte);
		MEMCPY(pAddrTo, adr2Byte, 8);
	ELSE
		MEMCPY( pAddrTo, pAddrFrom, nCurrentVarLength);
	END_IF
	
	(* Increment addressed of interest *)
	pAddrFrom := PAddrFrom + nCurrentVarLength;
	pAddrTo := pAddrTo + nCurrentVarLength;
END_FOR

END_FUNCTION

// ---- POUs/UR_TCP_IP_Data_Collection/F_FindAddr.TcPOU
FUNCTION F_FindAddr : POINTER TO BYTE
VAR_INPUT
	pAddrTo: POINTER TO BYTE;
	nByteCount: UINT;
END_VAR
VAR

END_VAR

IF nByteCount=8 THEN
	pAddrTo := pAddrTo;
	nByteCount := 0;
ELSIF nByteCount>8 THEN
	pAddrTo := pAddrTo + 16 - nByteCount;
	nByteCount := 0;
ELSE
	pAddrTo := pAddrTo;
END_IF

F_FindAddr := pAddrTo;

END_FUNCTION

// ---- POUs/UR_TCP_IP_Data_Collection/F_RecJointData.TcPOU
FUNCTION F_RecJointData : ST_JointData									// Different for different structures
VAR_INPUT
	data: ARRAY [1..500] OF BYTE;
END_VAR
VAR
	nNumOfVar: UINT;
	nIndex: UINT;
	pAddrTo: POINTER TO ST_JointData;
	PAddrFrom: POINTER TO ARRAY [1..500] OF BYTE;
	nByteCount: UINT;
	
	n2Byte : UINT;
	n4Byte : UDINT;
	n8Byte : ULINT;
	adr2Byte: POINTER TO UINT;
	adr4Byte: POINTER TO UDINT;
	adr8Byte: POINTER TO ULINT;
	nCurrentVarLength: USINT;
END_VAR

nNumOfVar := SIZEOF(F_RecJointData.arrVarLength);						// Different for different structures
pAddrTo := ADR(F_RecJointData);											// Different for different structures
PAddrFrom := ADR(data);
nByteCount := 0;
adr2Byte := ADR(n2Byte);
adr4Byte := ADR(n4Byte);
adr8Byte := ADR(n8Byte);

FOR nIndex := 1 TO nNumOfVar DO
	nCurrentVarLength := F_RecJointData.arrVarLength[nIndex];			// Different for different structures
	
	(* Determine byte address to save item to *)
	nByteCount := nByteCount + nCurrentVarLength;
	IF nByteCount=8 THEN
		pAddrTo := pAddrTo;
		nByteCount := 0;
	ELSIF nByteCount>8 THEN
		pAddrTo := pAddrTo + 16 - nByteCount;
		nByteCount := 0;
	ELSE
		pAddrTo := pAddrTo;
	END_IF
	
	(* Convert Data based on size of item (in bytes) *)
	IF nCurrentVarLength=8 THEN
		MEMCPY(adr8Byte, pAddrFrom, 8);
		n8Byte := BE64_TO_HOSTEX(n8Byte);
		MEMCPY(pAddrTo, adr8Byte, 8);
	ELSIF nCurrentVarLength=4 THEN
		MEMCPY(adr4Byte, pAddrFrom, 8);
		n4Byte := BE32_TO_HOST(n4Byte);
		MEMCPY(pAddrTo, adr4Byte, 8);
	ELSIF nCurrentVarLength=2 THEN
		MEMCPY(adr2Byte, pAddrFrom, 8);
		n2Byte := BE16_TO_HOST(n2Byte);
		MEMCPY(pAddrTo, adr2Byte, 8);
	ELSE
		MEMCPY( pAddrTo, pAddrFrom, nCurrentVarLength);
	END_IF
	
	(* Increment addressed of interest *)
	pAddrFrom := PAddrFrom + nCurrentVarLength;
	pAddrTo := pAddrTo + nCurrentVarLength;
END_FOR

END_FUNCTION

// ---- POUs/UR_TCP_IP_Data_Collection/F_RecCartesianInfo.TcPOU
FUNCTION F_RecCartesianInfo : ST_CartesianInfo								// Different for different structures
VAR_INPUT
	data: ARRAY [1..500] OF BYTE;
END_VAR
VAR
	nNumOfVar: UINT;
	nIndex: UINT;
	pAddrTo: POINTER TO ST_CartesianInfo;
	nAddrTo: POINTER TO ST_CartesianInfo;
	PAddrFrom: POINTER TO ARRAY [1..500] OF BYTE;
	nByteCount: UINT;
	
	n2Byte : UINT;
	n4Byte : UDINT;
	n8Byte : ULINT;
	adr2Byte: POINTER TO UINT;
	adr4Byte: POINTER TO UDINT;
	adr8Byte: POINTER TO ULINT;
	nCurrentVarLength: USINT;
END_VAR

nNumOfVar := SIZEOF(F_RecCartesianInfo.arrVarLength);						// Different for different structures
pAddrTo := ADR(F_RecCartesianInfo);											// Different for different structures
PAddrFrom := ADR(data);
adr2Byte := ADR(n2Byte);
adr4Byte := ADR(n4Byte);
adr8Byte := ADR(n8Byte);

FOR nIndex := 1 TO nNumOfVar DO
	nCurrentVarLength := F_RecCartesianInfo.arrVarLength[nIndex];			// Different for different structures
	
	(* Determine byte address to save item to *)
	nByteCount := nByteCount + nCurrentVarLength;
	IF nByteCount=8 THEN
		pAddrTo := pAddrTo;
		nByteCount := 0;
	ELSIF nByteCount>8 THEN
		pAddrTo := pAddrTo + 16 - nByteCount;
		nByteCount := 0;
	ELSE
		pAddrTo := pAddrTo;
	END_IF
	nAddrTo := F_FindAddr(pAddrTo,nByteCount);
	
	(* Convert Data based on size of item (in bytes) *)
	IF nCurrentVarLength=8 THEN
		MEMCPY(adr8Byte, pAddrFrom, 8);
		n8Byte := BE64_TO_HOSTEX(n8Byte);
		MEMCPY(pAddrTo, adr8Byte, 8);
	ELSIF nCurrentVarLength=4 THEN
		MEMCPY(adr4Byte, pAddrFrom, 8);
		n4Byte := BE32_TO_HOST(n4Byte);
		MEMCPY(pAddrTo, adr4Byte, 8);
	ELSIF nCurrentVarLength=2 THEN
		MEMCPY(adr2Byte, pAddrFrom, 8);
		n2Byte := BE16_TO_HOST(n2Byte);
		MEMCPY(pAddrTo, adr2Byte, 8);
	ELSE
		MEMCPY( pAddrTo, pAddrFrom, nCurrentVarLength);
	END_IF
	
	(* Increment addressed of interest *)
	pAddrFrom := PAddrFrom + nCurrentVarLength;
	pAddrTo := pAddrTo + nCurrentVarLength;
END_FOR

END_FUNCTION

// ---- POUs/UR_TCP_IP_Data_Collection/F_RecConfigurationData.TcPOU
FUNCTION F_RecConfigurationData : ST_ConfigurationData								// Different for different structures
VAR_INPUT
	data: ARRAY [1..500] OF BYTE;
END_VAR
VAR
	nNumOfVar: UINT;
	nIndex: UINT;
	pAddrTo: POINTER TO ST_ConfigurationData;										// Different for different structures
	PAddrFrom: POINTER TO ARRAY [1..500] OF BYTE;
	nByteCount: UINT;
	
	n2Byte : UINT;
	n4Byte : UDINT;
	n8Byte : ULINT;
	adr2Byte: POINTER TO UINT;
	adr4Byte: POINTER TO UDINT;
	adr8Byte: POINTER TO ULINT;
	nCurrentVarLength: USINT;
END_VAR

nNumOfVar := SIZEOF(F_RecConfigurationData.arrVarLength);						// Different for different structures
pAddrTo := ADR(F_RecConfigurationData);											// Different for different structures
PAddrFrom := ADR(data);
nByteCount := 0;
adr2Byte := ADR(n2Byte);
adr4Byte := ADR(n4Byte);
adr8Byte := ADR(n8Byte);

FOR nIndex := 1 TO nNumOfVar DO
	nCurrentVarLength := F_RecConfigurationData.arrVarLength[nIndex];			// Different for different structures
	
	(* Determine byte address to save item to *)
	nByteCount := nByteCount + nCurrentVarLength;
	IF nByteCount=8 THEN
		pAddrTo := pAddrTo;
		nByteCount := 0;
	ELSIF nByteCount>8 THEN
		pAddrTo := pAddrTo + 16 - nByteCount;
		nByteCount := 0;
	ELSE
		pAddrTo := pAddrTo;
	END_IF
	
	(* Convert Data based on size of item (in bytes) *)
	IF nCurrentVarLength=8 THEN
		MEMCPY(adr8Byte, pAddrFrom, 8);
		n8Byte := BE64_TO_HOSTEX(n8Byte);
		MEMCPY(pAddrTo, adr8Byte, 8);
	ELSIF nCurrentVarLength=4 THEN
		MEMCPY(adr4Byte, pAddrFrom, 8);
		n4Byte := BE32_TO_HOST(n4Byte);
		MEMCPY(pAddrTo, adr4Byte, 8);
	ELSIF nCurrentVarLength=2 THEN
		MEMCPY(adr2Byte, pAddrFrom, 8);
		n2Byte := BE16_TO_HOST(n2Byte);
		MEMCPY(pAddrTo, adr2Byte, 8);
	ELSE
		MEMCPY( pAddrTo, pAddrFrom, nCurrentVarLength);
	END_IF
	
	(* Increment addressed of interest *)
	pAddrFrom := PAddrFrom + nCurrentVarLength;
	pAddrTo := pAddrTo + nCurrentVarLength;
END_FOR

END_FUNCTION

// ---- POUs/UR_TCP_IP_Data_Collection/F_RecForceModeData.TcPOU
FUNCTION F_RecForceModeData : ST_ForceModeData								// Different for different structures
VAR_INPUT
	data: ARRAY [1..500] OF BYTE;
END_VAR
VAR
	nNumOfVar: UINT;
	nIndex: UINT;
	pAddrTo: POINTER TO ST_ForceModeData;
	nAddrTo: POINTER TO ST_ForceModeData;
	PAddrFrom: POINTER TO ARRAY [1..500] OF BYTE;
	nByteCount: UINT;
	
	n2Byte : UINT;
	n4Byte : UDINT;
	n8Byte : ULINT;
	adr2Byte: POINTER TO UINT;
	adr4Byte: POINTER TO UDINT;
	adr8Byte: POINTER TO ULINT;
	nCurrentVarLength: USINT;
END_VAR

nNumOfVar := SIZEOF(F_RecForceModeData.arrVarLength);						// Different for different structures
pAddrTo := ADR(F_RecForceModeData);											// Different for different structures
PAddrFrom := ADR(data);
adr2Byte := ADR(n2Byte);
adr4Byte := ADR(n4Byte);
adr8Byte := ADR(n8Byte);

FOR nIndex := 1 TO nNumOfVar DO
	nCurrentVarLength := F_RecForceModeData.arrVarLength[nIndex];			// Different for different structures
	
	(* Determine byte address to save item to *)
	nByteCount := nByteCount + nCurrentVarLength;
	IF nByteCount=8 THEN
		pAddrTo := pAddrTo;
		nByteCount := 0;
	ELSIF nByteCount>8 THEN
		pAddrTo := pAddrTo + 16 - nByteCount;
		nByteCount := 0;
	ELSE
		pAddrTo := pAddrTo;
	END_IF
	nAddrTo := F_FindAddr(pAddrTo,nByteCount);
	
	(* Convert Data based on size of item (in bytes) *)
	IF nCurrentVarLength=8 THEN
		MEMCPY(adr8Byte, pAddrFrom, 8);
		n8Byte := BE64_TO_HOSTEX(n8Byte);
		MEMCPY(pAddrTo, adr8Byte, 8);
	ELSIF nCurrentVarLength=4 THEN
		MEMCPY(adr4Byte, pAddrFrom, 8);
		n4Byte := BE32_TO_HOST(n4Byte);
		MEMCPY(pAddrTo, adr4Byte, 8);
	ELSIF nCurrentVarLength=2 THEN
		MEMCPY(adr2Byte, pAddrFrom, 8);
		n2Byte := BE16_TO_HOST(n2Byte);
		MEMCPY(pAddrTo, adr2Byte, 8);
	ELSE
		MEMCPY( pAddrTo, pAddrFrom, nCurrentVarLength);
	END_IF
	
	(* Increment addressed of interest *)
	pAddrFrom := PAddrFrom + nCurrentVarLength;
	pAddrTo := pAddrTo + nCurrentVarLength;
END_FOR

END_FUNCTION

// ---- POUs/FB_CSV_RobotDataWriter.TcPOU
FUNCTION_BLOCK FB_CSV_RobotDataWriter
VAR_INPUT
	bWriteLine:	BOOL;
	sFileName:	STRING;
	stRobotData : ST_UR;
	bEnable : BOOL;
END_VAR
VAR_OUTPUT
	bBusy:	BOOL;
	bFileOpen : BOOL;
	bError:	BOOL;
	sError:	STRING;
END_VAR
VAR
	fbFileOpen:	FB_FileOpen;
	fbFilePuts:	FB_FilePuts;
	fbFileClose:	FB_FileClose;
	
	rtWrite:	R_TRIG;
	
	nState:	INT;
	sTempPathName:	STRING;
	sDataString1:	STRING(255);
	sDataString2:	STRING(255);
	
	nLastTimestamp : LWORD;
END_VAR

//rtWrite(	CLK := bWriteLine);

CASE nState OF
	0:	(*IDLE*)
		bBusy := FALSE;
		// choose state		
		IF bFileOpen AND NOT bEnable THEN
			// close file
			nState := 30;
		END_IF
		
		IF nLastTimestamp <> stRobotData.RobotModeData.Timestamp THEN
			bWriteLine := FALSE;
			bBusy := TRUE;
			bError := FALSE;
			sError := '';
			sTempPathName := CONCAT(CONCAT('D:\PLCTempData\',sFileName),'.csv');
			// Build Datastrings
			// uint = 20 characters, word = 6 characters, bool = 5 characters, lword = 11, lreal = 16/15 
			// 12 ulints = 240 bytes max string length of 255
			sDataString1 := '';
			//time
			sDataString1 := INSERT(sDataString1,CONCAT(LWORD_TO_STRING(Global.nCurrentTime),','),LEN(sDataString1));
			sDataString1 := INSERT(sDataString1,CONCAT(LWORD_TO_STRING(stRobotData.RobotModeData.Timestamp),','),LEN(sDataString1));
			//position
			sDataString1 := INSERT(sDataString1,CONCAT(LREAL_TO_STRING(stRobotData.JointData.j1_qactual),','),LEN(sDataString1));
			sDataString1 := INSERT(sDataString1,CONCAT(LREAL_TO_STRING(stRobotData.JointData.j2_qactual),','),LEN(sDataString1));
			sDataString1 := INSERT(sDataString1,CONCAT(LREAL_TO_STRING(stRobotData.JointData.j3_qactual),','),LEN(sDataString1));
			sDataString1 := INSERT(sDataString1,CONCAT(LREAL_TO_STRING(stRobotData.JointData.j4_qactual),','),LEN(sDataString1));
			sDataString1 := INSERT(sDataString1,CONCAT(LREAL_TO_STRING(stRobotData.JointData.j5_qactual),','),LEN(sDataString1));
			sDataString1 := INSERT(sDataString1,CONCAT(LREAL_TO_STRING(stRobotData.JointData.j6_qactual),','),LEN(sDataString1));
			
			// Second half of part data
			sDataString2 := '';
			//velocity
			sDataString2 := INSERT(sDataString2,CONCAT(LREAL_TO_STRING(stRobotData.JointData.j1_qdactual),','),LEN(sDataString2));
			sDataString2 := INSERT(sDataString2,CONCAT(LREAL_TO_STRING(stRobotData.JointData.j2_qdactual),','),LEN(sDataString2));
			sDataString2 := INSERT(sDataString2,CONCAT(LREAL_TO_STRING(stRobotData.JointData.j3_qdactual),','),LEN(sDataString2));
			sDataString2 := INSERT(sDataString2,CONCAT(LREAL_TO_STRING(stRobotData.JointData.j4_qdactual),','),LEN(sDataString2));
			sDataString2 := INSERT(sDataString2,CONCAT(LREAL_TO_STRING(stRobotData.JointData.j5_qdactual),','),LEN(sDataString2));
			sDataString2 := INSERT(sDataString2,CONCAT(LREAL_TO_STRING(stRobotData.JointData.j6_qdactual),','),LEN(sDataString2));
			// Tool XYZ
			sDataString2 := INSERT(sDataString2,CONCAT(LREAL_TO_STRING(stRobotData.CartesianInfo.ToolX),','),LEN(sDataString2));
			sDataString2 := INSERT(sDataString2,CONCAT(LREAL_TO_STRING(stRobotData.CartesianInfo.ToolY),','),LEN(sDataString2));
			sDataString2 := INSERT(sDataString2,CONCAT(LREAL_TO_STRING(stRobotData.CartesianInfo.ToolZ),','),LEN(sDataString2));
			// New line
			sDataString2 := CONCAT(sDataString2,'$N');
			
			// Keep track of new messages
			nLastTimestamp := stRobotData.RobotModeData.Timestamp;
			
			// go to next state
			IF bFileOpen THEN
				// start writing strings
				nState := 20;
			ELSE
				// open file
				nState := 10;
			END_IF
		END_IF		
	
	10:	(*Open File*)	
		fbFileOpen(	sPathName := sTempPathName,
					nMode := FOPEN_MODEAPPEND,
					bExecute := TRUE,
					tTimeOut := T#1S);
		IF NOT fbFileOpen.bBusy THEN
			fbFileOpen(	bExecute := FALSE);
			IF fbFileOpen.bError THEN
				bError := TRUE;
				sError := 'Could Not Open File';
				nState := 0;
			ELSE
				bFileOpen := TRUE;
				nState := nState + 10;
			END_IF
		END_IF
		
	20:	(*Write Line To File*)
		fbFilePuts(	hFile := fbFileOpen.hFile,
					sLine := sDataString1,
					bExecute := TRUE,
					tTimeout := T#1S);
		IF NOT fbFilePuts.bBusy THEN
			fbFilePuts(	bExecute := FALSE);
			IF fbFilePuts.bError THEN
				bError := TRUE;
				sError := 'Could not write to file';
				nState := nState + 10;
			ELSE
				nState := nState + 1;
			END_IF
		END_IF
	21:	(*Write Line To File*)
		fbFilePuts(	hFile := fbFileOpen.hFile,
					sLine := sDataString2,
					bExecute := TRUE,
					tTimeout := T#1S);
		IF NOT fbFilePuts.bBusy THEN
			fbFilePuts(	bExecute := FALSE);
			IF fbFilePuts.bError THEN
				bError := TRUE;
				sError := 'Could not write to file';
				nState := 30;
			ELSE
				IF bEnable THEN
					nState := 0;
				ELSE
					nState := 30;
				END_IF
			END_IF
		END_IF
		
	30:	(*Close File*)
		fbFileClose(	hFile := fbFileOpen.hFile,
						bExecute := TRUE,
						tTimeout := T#1S);
		IF NOT fbFileClose.bBusy THEN
			fbFileClose(	bExecute := FALSE);
			IF fbFileClose.bError THEN
				bError := TRUE;
				sError := 'Could not close file';
				nState := 0;
			ELSE
				bFileOpen := FALSE;
				nState := 0;
			END_IF
		END_IF
END_CASE

END_FUNCTION_BLOCK

// ---- POUs/FB_FT_UDPConnection.TcPOU
FUNCTION_BLOCK FB_FT_UDPConnection
VAR_INPUT
	bEnable : BOOL;
	Robot : STRING;
	bRecordData : BOOL;
	
END_VAR
VAR_OUTPUT
	bBusy : BOOL;
	bConnected : BOOL;
	bInitialized : BOOL;
	bError : BOOL;
	stOptoforceData : ST_OptoforceUDPData;
END_VAR
VAR
	stRequest : ST_OptoforceUDPRequest := (Header := 4660, Command := 2, Data := 0);
	fbConnectionlessSocket : FB_ConnectionlessSocket;
	fbSocketUdpCreate : FB_SocketUdpCreate := (sSrvNetId := '', tTimeout := DEFAULT_ADS_TIMEOUT);
	fbSocketUdpSendTo : FB_SocketUdpSendTo := (sSrvNetId := '', tTimeout := DEFAULT_ADS_TIMEOUT);
	fbSocketUdpReceiveFrom : FB_SocketUdpReceiveFrom := (sSrvNetId := '', tTimeout := DEFAULT_ADS_TIMEOUT);
	fbSocketClose : FB_SocketClose := (sSrvNetId := '', tTimeout := DEFAULT_ADS_TIMEOUT);
	eState : E_UDPConnection;
	hSocket : T_HSOCKET;
	receivebuffer : ARRAY [1..9] OF UDINT;
	sendbuffer : ST_OptoforceUDPRequest;
	index: INT;
	fbRecordFTData : FB_CSV_FTDataWriter;
END_VAR

CASE eState OF
	E_UDPConnection.Idle:
		IF bEnable THEN
			bBusy := TRUE;
			IF NOT bConnected THEN
				eState := E_UDPConnection.Connect_Start;
			ELSIF NOT bInitialized THEN
				eState := E_UDPConnection.Request_Start;
			ELSE
				eState := E_UDPConnection.Receive_Start;
			END_IF
		ELSIF bConnected THEN
			eState := E_UDPConnection.Close_Start;
		END_IF
	E_UDPConnection.Connect_Start:
		fbSocketUdpCreate.bExecute := TRUE;
		//fbSocketUdpCreate.nLocalPort := 200;
		eState := E_UDPConnection.Connect_Wait;
	E_UDPConnection.Connect_Wait:
		fbSocketUdpCreate.bExecute := FALSE;
		IF fbSocketUdpCreate.bError THEN
			eState := E_UDPConnection.HandleError;
		ELSIF NOT fbSocketUdpCreate.bBusy THEN
			bConnected := TRUE;
			hSocket := fbSocketUdpCreate.hSocket;
			eState := E_UDPConnection.Idle;
		END_IF
	E_UDPConnection.Request_Start:
		sendbuffer.Command := HOST_TO_BE16(stRequest.Command);
		sendbuffer.Header := HOST_TO_BE16(stRequest.Header);
		sendbuffer.Data := HOST_TO_BE32(stRequest.Data);
	
		fbSocketUdpSendTo.bExecute := TRUE;
		fbSocketUdpSendTo.hSocket := hSocket;
		
		fbSocketUdpSendTo.pSrc := ADR(sendbuffer);
		fbSocketUdpSendTo.cbLen := SIZEOF(sendbuffer);
		
		fbSocketUdpSendTo.sRemoteHost := '192.168.1.1';
		fbSocketUdpSendTo.nRemotePort := 49152;
		
		eState := E_UDPConnection.Request_Wait;
		
	E_UDPConnection.Request_Wait:
		fbSocketUdpSendTo.bExecute := FALSE;
		
		IF fbSocketUdpSendTo.bError THEN
			eState := E_UDPConnection.HandleError;
		ELSIF NOT fbSocketUdpSendTo.bBusy THEN
			bInitialized := TRUE;
			eState := E_UDPConnection.Idle;
		END_IF
		
	E_UDPConnection.Receive_Start:
		fbSocketUdpReceiveFrom.bExecute := TRUE;
		fbSocketUdpReceiveFrom.hSocket := hSocket;
		
		fbSocketUdpReceiveFrom.cbLen := SIZEOF(receivebuffer);
		fbSocketUdpReceiveFrom.pDest := ADR(receivebuffer);
		
		eState := E_UDPConnection.Receive_Wait;
		
	E_UDPConnection.Receive_Wait:
		fbSocketUdpReceiveFrom.bExecute := FALSE;
		IF fbSocketUdpReceiveFrom.bError THEN
			eState := E_UDPConnection.HandleError;
		ELSIF NOT fbSocketUdpReceiveFrom.bBusy THEN
			IF fbSocketUdpReceiveFrom.nRecBytes=36 THEN
				FOR index:=1 TO 9 DO
					receivebuffer[index] := BE32_TO_HOST(receivebuffer[index]);
				END_FOR
				MEMCPY(srcAddr := ADR(receivebuffer), destAddr := ADR(stOptoforceData), n := 36);
				(*// Do data conversion to Newtons and N-m
				stOptoforceData.Fx := stOptoforceData.Fx/10000;
				stOptoforceData.Fy := stOptoforceData.Fy/10000;
				stOptoforceData.Fz := stOptoforceData.Fz/10000;
				stOptoforceData.Tx := stOptoforceData.Tx/100000;
				stOptoforceData.Ty := stOptoforceData.Ty/100000;
				stOptoforceData.Tz := stOptoforceData.Tz/100000;
				*)
				IF bRecordData THEN
					eState := E_UDPConnection.RecordData;
				ELSE
					eState := E_UDPConnection.Idle;
				END_IF
			ELSE
				eState := E_UDPConnection.Idle;
			END_IF
		END_IF
		
	E_UDPConnection.RecordData:
		fbRecordFTData.bEnable := TRUE;
		fbRecordFTData.sFileName := 'FTData';
		fbRecordFTData.stFTData := stOptoforceData;
		IF NOT fbRecordFTData.bBusy THEN
			eState := E_UDPConnection.Idle;
		END_IF
		
	E_UDPConnection.Close_Start:
		fbSocketClose.bExecute := TRUE;
		fbSocketClose.hSocket := hSocket;
		
		eState := E_UDPConnection.Close_Wait;
	
	E_UDPConnection.Close_Wait:
		fbSocketClose.bExecute := FALSE;
		IF fbSocketClose.bError THEN
				eState := E_UDPConnection.HandleError;
		ELSIF NOT fbSocketClose.bBusy THEN
			MEMSET(ADR(hSocket),0,SIZEOF(hSocket));
			bBusy := FALSE;
			bConnected := FALSE;
			bInitialized := FALSE;
			bError := FALSE;
			eState := E_UDPConnection.Idle;
		END_IF
		
	E_UDPConnection.HandleError:
		eState := E_UDPConnection.Close_Start;
END_CASE

fbSocketUdpCreate();
fbConnectionlessSocket();
fbSocketUdpSendTo();
fbSocketUdpReceiveFrom();
fbSocketClose();
fbRecordFTData();

END_FUNCTION_BLOCK

// ---- POUs/FB_CSV_FTDataWriter.TcPOU
FUNCTION_BLOCK FB_CSV_FTDataWriter
VAR_INPUT
	bWriteLine : BOOL;
	sFileName:	STRING;
	stFTData : ST_OptoforceUDPData;
	bEnable : BOOL;
END_VAR
VAR_OUTPUT
	bBusy:	BOOL;
	bFileOpen : BOOL;
	bError:	BOOL;
	sError:	STRING;
END_VAR
VAR
	fbFileOpen:	FB_FileOpen;
	fbFilePuts:	FB_FilePuts;
	fbFileClose:	FB_FileClose;
	
	rtWrite:	R_TRIG;
	
	nState:	INT;
	sTempPathName:	STRING;
	sDataString1:	STRING(255);
	sDataString2:	STRING(255);
	
	nLastTimestamp : UDINT;
END_VAR

//rtWrite(	CLK := bWriteLine);

CASE nState OF
	0:	(*IDLE*)
		bBusy := FALSE;
		// choose state		
		IF bFileOpen AND NOT bEnable THEN
			// close file
			nState := 30;
		END_IF
		
		IF nLastTimestamp <> stFTData.FT_sequence THEN
			bWriteLine := FALSE;
			bBusy := TRUE;
			bError := FALSE;
			sError := '';
			sTempPathName := CONCAT(CONCAT('D:\PLCTempData\',sFileName),'.csv');
			// Build Datastrings
			// uint = 20 characters, word = 6 characters, bool = 5 characters, lword = 11, lreal = 16/15 
			// 12 ulints = 240 bytes max string length of 255
			sDataString1 := '';
			//time
			sDataString1 := INSERT(sDataString1,CONCAT(LWORD_TO_STRING(Global.nCurrentTime),','),LEN(sDataString1));
			sDataString1 := INSERT(sDataString1,CONCAT(UDINT_TO_STRING(stFTData.FT_sequence),','),LEN(sDataString1));
			//position
			sDataString1 := INSERT(sDataString1,CONCAT(DINT_TO_STRING(stFTData.HS_sequence),','),LEN(sDataString1));
			sDataString1 := INSERT(sDataString1,CONCAT(DINT_TO_STRING(stFTData.Status),','),LEN(sDataString1));
			sDataString1 := INSERT(sDataString1,CONCAT(DINT_TO_STRING(stFTData.Fx),','),LEN(sDataString1));
			sDataString1 := INSERT(sDataString1,CONCAT(DINT_TO_STRING(stFTData.Fy),','),LEN(sDataString1));
			sDataString1 := INSERT(sDataString1,CONCAT(DINT_TO_STRING(stFTData.Fz),','),LEN(sDataString1));
			sDataString1 := INSERT(sDataString1,CONCAT(DINT_TO_STRING(stFTData.Tx),','),LEN(sDataString1));
			sDataString1 := INSERT(sDataString1,CONCAT(DINT_TO_STRING(stFTData.Ty),','),LEN(sDataString1));
			sDataString1 := INSERT(sDataString1,CONCAT(DINT_TO_STRING(stFTData.Tz),','),LEN(sDataString1));
			sDataString1 := CONCAT(sDataString1,'$N');
			
			(*
			// Second half of part data
			sDataString2 := '';
			//velocity
			sDataString2 := INSERT(sDataString2,CONCAT(LREAL_TO_STRING(stRobotData.JointData.j1_qdactual),','),LEN(sDataString2));
			sDataString2 := INSERT(sDataString2,CONCAT(LREAL_TO_STRING(stRobotData.JointData.j2_qdactual),','),LEN(sDataString2));
			sDataString2 := INSERT(sDataString2,CONCAT(LREAL_TO_STRING(stRobotData.JointData.j3_qdactual),','),LEN(sDataString2));
			sDataString2 := INSERT(sDataString2,CONCAT(LREAL_TO_STRING(stRobotData.JointData.j4_qdactual),','),LEN(sDataString2));
			sDataString2 := INSERT(sDataString2,CONCAT(LREAL_TO_STRING(stRobotData.JointData.j5_qdactual),','),LEN(sDataString2));
			sDataString2 := INSERT(sDataString2,CONCAT(LREAL_TO_STRING(stRobotData.JointData.j6_qdactual),','),LEN(sDataString2));
			// Tool XYZ
			sDataString2 := INSERT(sDataString2,CONCAT(LREAL_TO_STRING(stRobotData.CartesianInfo.ToolX),','),LEN(sDataString2));
			sDataString2 := INSERT(sDataString2,CONCAT(LREAL_TO_STRING(stRobotData.CartesianInfo.ToolY),','),LEN(sDataString2));
			sDataString2 := INSERT(sDataString2,CONCAT(LREAL_TO_STRING(stRobotData.CartesianInfo.ToolZ),','),LEN(sDataString2));
			// New line
			sDataString2 := CONCAT(sDataString2,'$N');
			*)
			
			// Keep track of new messages
			nLastTimestamp := stFTData.FT_sequence;
			
			// go to next state
			IF bFileOpen THEN
				// start writing strings
				nState := 20;
			ELSE
				// open file
				nState := 10;
			END_IF
		END_IF		
	
	10:	(*Open File*)	
		fbFileOpen(	sPathName := sTempPathName,
					nMode := FOPEN_MODEAPPEND,
					bExecute := TRUE,
					tTimeOut := T#1S);
		IF NOT fbFileOpen.bBusy THEN
			fbFileOpen(	bExecute := FALSE);
			IF fbFileOpen.bError THEN
				bError := TRUE;
				sError := 'Could Not Open File';
				nState := 0;
			ELSE
				bFileOpen := TRUE;
				nState := nState + 10;
			END_IF
		END_IF
		
	20:	(*Write Line To File*)
		fbFilePuts(	hFile := fbFileOpen.hFile,
					sLine := sDataString1,
					bExecute := TRUE,
					tTimeout := T#1S);
		IF NOT fbFilePuts.bBusy THEN
			fbFilePuts(	bExecute := FALSE);
			IF fbFilePuts.bError THEN
				bError := TRUE;
				sError := 'Could not write to file';
				nState := nState + 10;
			ELSE
				nState := nState + 10; // make +1 for second string inclusion
			END_IF
		END_IF
	21:	(*Write Line To File*)
		fbFilePuts(	hFile := fbFileOpen.hFile,
					sLine := sDataString2,
					bExecute := TRUE,
					tTimeout := T#1S);
		IF NOT fbFilePuts.bBusy THEN
			fbFilePuts(	bExecute := FALSE);
			IF fbFilePuts.bError THEN
				bError := TRUE;
				sError := 'Could not write to file';
				nState := 30;
			ELSE
				IF bEnable THEN
					nState := 0;
				ELSE
					nState := 30;
				END_IF
			END_IF
		END_IF
		
	30:	(*Close File*)
		fbFileClose(	hFile := fbFileOpen.hFile,
						bExecute := TRUE,
						tTimeout := T#1S);
		IF NOT fbFileClose.bBusy THEN
			fbFileClose(	bExecute := FALSE);
			IF fbFileClose.bError THEN
				bError := TRUE;
				sError := 'Could not close file';
				nState := 0;
			ELSE
				bFileOpen := FALSE;
				nState := 0;
			END_IF
		END_IF
END_CASE

END_FUNCTION_BLOCK

// ---- POUs/P_Safety.TcPOU
PROGRAM P_Safety
VAR

	UR5Mode_pointer: POINTER TO BYTE;
	UR5Mode: WORD;
	mbReadUR5Mode : FB_mbReadRegs;
	UR5Mode2: WORD;
	
	blinker: TON := (PT := T#500MS);
	
	fbUR5mode : FB_mbReadSingleReg;
	fbUR3mode : FB_mbReadSingleReg;
END_VAR

// Handle Acknoledging Error and Reseting Safety PLC
Global_Safety.ErrorAck := Global_Safety.ResetPB;

// Get mode from UR5
fbUR5Mode(	Robot := 'UR5',
			Register := Global.ModeAddr);
Global.stUR5.mode := fbUR5Mode.Value;

// Get mode from UR3
fbUR3Mode(	Robot := 'UR3',
			Register := Global.ModeAddr);
Global.stUR3.mode := fbUR3Mode.Value;

// Monitor Robot Status for Stack Lights
// RED - Robots Enabled (mode = 7)
IF Global.stUR3.mode=7 THEN
	Global_Safety.UR3RedIND := TRUE;
ELSE
	Global_Safety.UR3RedIND := FALSE;
END_IF
IF Global.stUR5.mode=7 THEN
	Global_Safety.UR5RedIND := TRUE;
ELSE
	Global_Safety.UR5RedIND := FALSE;
END_IF


// AMBER - Safeguard Fault
IF NOT Global_Safety.NotInEStop OR NOT Global_Safety.NotInRedSpeed OR NOT Global_Safety.NotInSafeStop THEN
	Global_Safety.UR3AmberIND := TRUE;
	Global_Safety.UR5AmberIND := TRUE;
ELSE
	Global_Safety.UR3AmberIND := FALSE;
	Global_Safety.UR5AmberIND := FALSE;
	// Control Pendant Indicator
	Global_Safety.CPFaultIND := FALSE; // if no faults turn off fault indicator
END_IF

// GREEN - Safety Systems On
IF Global_Safety.SafetyPLCState=1 THEN
	Global_Safety.UR3GreenIND := TRUE;
	Global_Safety.UR5GreenIND := TRUE;
ELSE
	Global_Safety.UR3GreenIND := FALSE;
	Global_Safety.UR5GreenIND := FALSE;
END_IF

// BLUE - Some Safety Systems Disabled
IF Global_Safety.ProgramModeActive THEN
	Global_Safety.UR3BlueIND := TRUE;
	Global_Safety.UR5BlueIND := TRUE;
	// Control Pendant 
	Global_Safety.CPEProgramModeIND := TRUE;
ELSE
	Global_Safety.UR3BlueIND := FALSE;
	Global_Safety.UR5BlueIND := FALSE;
	// Control Pendant 
	Global_Safety.CPEProgramModeIND := FALSE;
END_IF

// Control Pendant Indicators
IF NOT Global_Safety.NotInEStop THEN // if in estop
	Global_Safety.CPEStopIND := TRUE; // turn on estop indicator
	blinker(IN := NOT blinker.Q); // blink reset light
	IF blinker.Q THEN // if timer went off and fault indicator not on 
		Global_Safety.CPFaultIND := NOT Global_Safety.CPFaultIND; // turn on fault indicator
	END_IF
ELSE // if not in estop
	Global_Safety.CPEStopIND := FALSE; // turn off estop indicator
	IF NOT Global_Safety.NotInRedSpeed OR NOT Global_Safety.NotInSafeStop THEN
		Global_Safety.CPFaultIND := TRUE; // if safe stop or red speed faults turn on fault indicator solid
	END_IF
END_IF

END_PROGRAM

// ---- POUs/Modbus POUs/FB_mbReadSingleReg.TcPOU
FUNCTION_BLOCK FB_mbReadSingleReg
VAR_INPUT
	Robot : STRING;
	Register : UINT;
END_VAR
VAR_OUTPUT
	Value : WORD;
END_VAR
VAR
	mbRead : FB_mbReadRegs;
	state : int;
END_VAR

(* 
FB_mbReadSingleReg - Function Block that can be called to read a single MODBUS register from a pre-defined UR Robot
	INPUTS:
		- Robot: 'UR5' or 'UR3'
		- Register: register number to read
	OUTPUTS
		- Value: The returned value
*)

// Set function block vairables
mbRead.nQuantity := 1;
mbRead.cbLength := 2;

IF Robot='UR5' THEN
	mbRead.sIPAddr := Global.stUR5.IP;
	mbRead.nTCPPort := Global.stUR5.mbPort;
	mbRead.nUnitID := Global.stUR5.unitID;
ELSIF Robot='UR3' THEN
	mbRead.sIPAddr := Global.stUR3.IP;
	mbRead.nTCPPort := Global.stUR3.mbPort;
	mbRead.nUnitID := Global.stUR3.unitID;
END_IF

mbRead.pDestAddr := ADR(Value);
mbRead.nMBAddr := Register;

// Set/Determine State of Function block
CASE state OF
	0:
		mbRead.bExecute := TRUE;
		state := 10;
	10:
		IF NOT mbRead.bBusy THEN
			mbRead.bExecute :=FALSE;
			state := 0;
		END_IF
END_CASE

// Run function block
mbRead();

END_FUNCTION_BLOCK

// ---- POUs/P_InputOutputHandling.TcPOU
PROGRAM P_InputOutputHandling
VAR
	// User Inputs
	// Process Selection
	nProcessType : INT := 1; // 1 = continuous, 2 = batch
	sProcessType : STRING := 'Continuous';
	bSwitchProcess : BOOL;
	
	bAutoLoad : BOOL;
	bAutoUnload : BOOL := TRUE;
	
	// Continuous Process
	InputTimer : TON;
	OutputTimer : TON;
	
	// Batch Process
	nBatchSize : INT := 1;
	
	// Loading and Unloading
	bRemoveParts : BOOL;
	bAddParts : BOOL;
	nInputIndex : INT;
	nOutputIndex : INT;
	
	// Data Recording
	fbPartRecordWriter:	FB_CSV_PartDataWriter;
	stLastPart : ST_Part;
	bWriteLine:	BOOL;
	sPartDataFileName:	STRING :='PartData';
END_VAR

(* =======================================================
Process Type Selection/Switching
======================================================= *)
IF bSwitchProcess THEN
	bSwitchProcess := FALSE;
	IF nProcessType = 1 THEN
		nProcessType := 2;
		sProcessType := 'Batch';
	ELSIF nProcessType = 2 THEN
		nProcessType := 1;
		sProcessType := 'Continuous';
	END_IF
END_IF

CASE nProcessType OF
	// Continuous Process
	1:	
		nBatchSize := 1;
		Global.nNumInputFixtures := nBatchSize;
		Global.nNumOutputFixtures := nBatchSize;
		
		// Refilling Input 
		IF bAutoLoad THEN
			// TODO replace this portion of code with a prenense detention sensor
			// to indicate a part available at the input
			InputTimer(IN := NOT Global.arrInputFixtures[1].stPart.bExists, PT := T#5S);
			IF InputTimer.Q THEN
				bAddParts := TRUE;
			END_IF
		END_IF
		IF bAutoUnload THEN
			// Emptying Output
			OutputTimer(IN := Global.arrOutputFixtures[1].stPart.bExists, PT := T#3S);
			IF OutputTimer.Q THEN
				bRemoveParts := TRUE;			
			END_IF
		END_IF
	// Batch Process
	2:
	// TODO batch process loading and unloading
	Global.nNumInputFixtures := nBatchSize;
	Global.nNumOutputFixtures := nBatchSize;
	
	
END_CASE

(* =======================================================
Adding and Removing Parts from WorkCell
======================================================= *)
IF bAddParts THEN
	FOR nInputIndex := 1 TO Global.nNumInputFixtures DO
		IF NOT Global.arrInputFixtures[1].stPart.bExists THEN
			Global.arrInputFixtures[nInputIndex].stPart.ntPartAdded := Global.nCurrentTime;
			Global.arrInputFixtures[nInputIndex].stPart.rtUR3TimePartAdded := Global.stUR3.RobotModeData.Timestamp;
			Global.arrInputFixtures[nInputIndex].stPart.rtUR5TimePartAdded := Global.stUR5.RobotModeData.Timestamp;
			Global.arrInputFixtures[nInputIndex].stPart.bExists := TRUE;
			Global.nPartsStarted := Global.nPartsStarted + 1;
			Global.arrInputFixtures[nInputIndex].stPart.nPartNumber := Global.nPartsStarted;
			bAddParts := FALSE;
		END_IF
	END_FOR
END_IF

IF bRemoveParts THEN
	FOR nOutputIndex := 1 TO Global.nNumOutputFixtures DO
		IF Global.arrOutputFixtures[nOutputIndex].stPart.bExists THEN
			Global.arrOutputFixtures[nOutputIndex].stPart.ntPartRemoved := Global.nCurrentTime;	
		
			// Record Part being removed
			stLastPart := Global.arrOutputFixtures[nOutputIndex].stPart;
			bWriteLine := TRUE; // initiate csv writer
			
			// Log times
			Global.nTotalPartTime := Global.nTotalPartTime + (stLastPart.ntPartRemoved - stLastPart.ntPartAdded);
			IF Global.nPartsCompleted > 0 THEN
				Global.nAveragePartTime := ULINT_TO_LREAL((Global.nTotalPartTime / Global.nPartsCompleted))/10000000;
			ELSE
				Global.nAveragePartTime := ULINT_TO_LREAL(Global.nTotalPartTime)/10000000;
			END_IF
			
			Global.nPartsCompleted := Global.nPartsCompleted + 1;
			
			// Log in internal log for visualization
			MEMMOVE(destAddr := ADR(Global.CompletedParts[2]),srcAddr := ADR(Global.CompletedParts), n:= SIZEOF(stLastPart)*9);
			MEMMOVE(destAddr := ADR(Global.CompletedParts[1]),srcAddr := ADR(stLastPart), n:= SIZEOF(stLastPart));
			Global.arrOutputFixtures[nOutputIndex].stPart := Global.stNullPart;
			
			// Pos Check Part Counting
			// Global.nPartsSincePosCheck := Global.nPartsSincePosCheck + 1;
			
		END_IF
	END_FOR
	bRemoveParts := FALSE;
END_IF

// TODO: make this work in batch mode. Currently will only record last part in for loop

fbPartRecordWriter.bEnable := Global.bActivatePartDataRecording; 
fbPartRecordWriter(	sFileName := sPartDataFileName,
					stPartData := stLastPart);
bWriteLine := FALSE;

END_PROGRAM

// ---- POUs/FB_CSV_PartDataWriter.TcPOU
FUNCTION_BLOCK FB_CSV_PartDataWriter
VAR_INPUT
	bEnable: BOOL;
	sFileName:	STRING;
	stPartData : ST_Part;
END_VAR
VAR_OUTPUT
	bBusy:	BOOL;
	bError:	BOOL;
	sError:	STRING;
END_VAR
VAR
	fbFileOpen:	FB_FileOpen;
	fbFilePuts:	FB_FilePuts;
	fbFileClose:	FB_FileClose;
	
	rtWrite:	R_TRIG;
	
	nState:	INT;
	sTempPathName:	STRING;
	sDataString1:	STRING(255);
	sDataString2:	STRING(255);
	bFileOpen: BOOL;
	
	nLastPart: WORD;
END_VAR

CASE nState OF
	0:	(*IDLE*)
		bBusy := FALSE;
		// choose state		
		IF bFileOpen AND NOT bEnable THEN
			// close file
			nState := 30;
		END_IF
		
		IF nLastPart <> stPartData.nPartNumber THEN

			sTempPathName := CONCAT(CONCAT('D:\PLCTempData\',sFileName),'.csv');
			// Build Datastrings
			// uint = 20 characters, word = 6 characters, bool = 5 characters, lword = 11
			// 12 ulints = 240 bytes max string length of 255
			sDataString1 := '';
			sDataString1 := INSERT(sDataString1,CONCAT(WORD_TO_STRING(stPartData.nPartNumber),','),LEN(sDataString1));
			sDataString1 := INSERT(sDataString1,CONCAT(WORD_TO_STRING(stPartData.nWorkFixture),','),LEN(sDataString1));
			sDataString1 := INSERT(sDataString1,CONCAT(WORD_TO_STRING(stPartData.nInputPosition),','),LEN(sDataString1));
			sDataString1 := INSERT(sDataString1,CONCAT(WORD_TO_STRING(stPartData.nOutputPosition),','),LEN(sDataString1));
			sDataString1 := INSERT(sDataString1,CONCAT(WORD_TO_STRING(stPartData.nPartType),','),LEN(sDataString1));
			sDataString1 := INSERT(sDataString1,CONCAT(BOOL_TO_STRING(stPartData.bComplete),','),LEN(sDataString1));
			sDataString1 := INSERT(sDataString1,CONCAT(LWORD_TO_STRING(stPartData.rtUR3TimePartAdded),','),LEN(sDataString1));
			sDataString1 := INSERT(sDataString1,CONCAT(LWORD_TO_STRING(stPartData.rtUR5TimePartAdded),','),LEN(sDataString1));
			sDataString1 := INSERT(sDataString1,CONCAT(ULINT_TO_STRING(stPartData.ntPartAdded),','),LEN(sDataString1));
 			sDataString1 := INSERT(sDataString1,CONCAT(ULINT_TO_STRING(stPartData.ntPickFromInputAssigned),','),LEN(sDataString1));
			sDataString1 := INSERT(sDataString1,CONCAT(ULINT_TO_STRING(stPartData.ntInputPartPicked),','),LEN(sDataString1));
			sDataString1 := INSERT(sDataString1,CONCAT(ULINT_TO_STRING(stPartData.ntInputPartPlaced),','),LEN(sDataString1));
			sDataString1 := INSERT(sDataString1,CONCAT(ULINT_TO_STRING(stPartData.ntPlaceInWFComplete),','),LEN(sDataString1));
			sDataString1 := INSERT(sDataString1,CONCAT(ULINT_TO_STRING(stPartData.ntTaskAssigned),','),LEN(sDataString1));
			sDataString1 := INSERT(sDataString1,CONCAT(ULINT_TO_STRING(stPartData.ntTaskActionStart),','),LEN(sDataString1));
			
			
			// Second half of part data
			sDataString2 := '';
			sDataString2 := INSERT(sDataString2,CONCAT(ULINT_TO_STRING(stPartData.ntTaskActionComplete),','),LEN(sDataString2));
			sDataString2 := INSERT(sDataString2,CONCAT(ULINT_TO_STRING(stPartData.ntTaskComplete),','),LEN(sDataString2));
			sDataString2 := INSERT(sDataString2,CONCAT(ULINT_TO_STRING(stPartData.ntPickFromWFAssigned),','),LEN(sDataString2));
			sDataString2 := INSERT(sDataString2,CONCAT(ULINT_TO_STRING(stPartData.ntOutputPartPicked),','),LEN(sDataString2));
			sDataString2 := INSERT(sDataString2,CONCAT(ULINT_TO_STRING(stPartData.ntOutputPartPlaced),','),LEN(sDataString2));
			sDataString2 := INSERT(sDataString2,CONCAT(ULINT_TO_STRING(stPartData.ntPlaceInOutputComplete),','),LEN(sDataString2));
			sDataString2 := INSERT(sDataString2,CONCAT(ULINT_TO_STRING(stPartData.ntPartRemoved),','),LEN(sDataString2));
			sDataString2 := CONCAT(sDataString2,'$N');
			
			
			// Keep track of new messages
			nLastPart := stPartData.nPartNumber;
			
			// go to next state
			IF bFileOpen THEN
				// start writing strings
				nState := 20;
			ELSE
				// open file
				nState := 10;
			END_IF
		END_IF	
		
		// set variables
		bError := FALSE;
		sError := '';	
	
	10:	(*Open File*)	
		fbFileOpen(	sPathName := sTempPathName,
					nMode := FOPEN_MODEAPPEND,
					bExecute := TRUE,
					tTimeOut := T#1S);
		IF NOT fbFileOpen.bBusy THEN
			fbFileOpen(	bExecute := FALSE);
			IF fbFileOpen.bError THEN
				bError := TRUE;
				sError := 'Could Not Open File';
				nState := 0;
			ELSE
				nState := nState + 10;
			END_IF
		END_IF
		
	20:	(*Write Line To File*)
		fbFilePuts(	hFile := fbFileOpen.hFile,
					sLine := sDataString1,
					bExecute := TRUE,
					tTimeout := T#1S);
		IF NOT fbFilePuts.bBusy THEN
			fbFilePuts(	bExecute := FALSE);
			IF fbFilePuts.bError THEN
				bError := TRUE;
				sError := 'Could not write to file';
				nState := nState + 10;
			ELSE
				nState := nState + 1;
			END_IF
		END_IF
	21:	(*Write Line To File*)
		fbFilePuts(	hFile := fbFileOpen.hFile,
					sLine := sDataString2,
					bExecute := TRUE,
					tTimeout := T#1S);
		IF NOT fbFilePuts.bBusy THEN
			fbFilePuts(	bExecute := FALSE);
			IF fbFilePuts.bError THEN
				bError := TRUE;
				sError := 'Could not write to file';
				nState := 30;
			ELSE
				nState := 30;
			END_IF
		END_IF
		
	30:	(*Close File*)
		fbFileClose(	hFile := fbFileOpen.hFile,
						bExecute := TRUE,
						tTimeout := T#1S);
		IF NOT fbFileClose.bBusy THEN
			fbFileClose(	bExecute := FALSE);
			IF fbFileClose.bError THEN
				bError := TRUE;
				sError := 'Could not close file';
				nState := 0;
			ELSE
				nState := 0;
			END_IF
		END_IF
END_CASE

END_FUNCTION_BLOCK

// ---- POUs/P_TaskHandling.TcPOU
PROGRAM P_TaskHandling
VAR
	// Robot task status informaiton
	// UR3
	fbUR3TaskStatusInfo : FB_mbReadRobotTaskStatusInfo := (Robot := 'UR3');
	stUR3TaskStatus : ST_RobotTaskStatusInfo;
	// UR5
	fbUR5TaskStatusInfo : FB_mbReadRobotTaskStatusInfo := (Robot := 'UR5');
	stUR5TaskStatus : ST_RobotTaskStatusInfo;
	
	// Task Triggers
	StopAssignment_ftrig : F_TRIG;
	// UR3
	UR3TaskActive_rtrig : R_TRIG; // Task assigned (including positioning movements)
	UR3TaskComplete_ftrig : F_TRIG; // Task reported complete
	UR3ActionStart_rtrig : R_TRIG; // robot positioning for task over, part interaction begins
	UR3ActionComplete_ftrig : F_TRIG; // part interaction ends
	//UR5
	UR5TaskActive_rtrig : R_TRIG; // Task assigned (including positioning movements)
	UR5TaskComplete_ftrig : F_TRIG; // Task reported complete
	UR5ActionStart_rtrig : R_TRIG; // robot positioning for task over, part interaction begins
	UR5ActionComplete_ftrig : F_TRIG; // part interaction ends
	
	// General use indexes and counters
	nMaxTimeInWF : REAL;
	nWorkFixtureIndex : INT;
	nInputFixtureIndex : INT;
	nOutputFixtureIndex : INT;
	
	// UR3 Task State Macine
	eUR3TaskState : E_RobotTaskStates;
	
	// UR3 Active Task Targets
	nUR3TargetWorkFixtureIndex : INT;
	nUR3TargetWorkframe : WORD;
	nUR3TargetTask : WORD;
	nUR3TargetPart : WORD;
	
	// UR5 Task State Macine
	eUR5TaskState : E_RobotTaskStates;
	
	// UR5 Active Task Targets
	nUR5TargetWorkFixtureIndex : INT;
	nUR5TargetInputFixtureIndex : INT;
	nUR5TargetOutputFixtureIndex : INT;
	nUR5TargetPickFrame : WORD;
	nUR5TargetPlaceFrame : WORD;
	nUR5TargetTask: WORD; // 1 for input 2 for output
	sUR5TargetTask: STRING;
	nUR5TargetPart : WORD;
	
	// Task writing functionblocks
	fbWriteUR3Task : FB_mbWriteRobotTask := (Robot := 'UR3');
	fbWriteUR5Task : FB_mbWriteRobotTask := (Robot := 'UR5');
	fbUR3Resume : FB_mbWriteSingleReg := (Robot := 'UR3', Register := 145, Value := 1);
	fbUR5Resume : FB_mbWriteSingleReg := (Robot := 'UR5', Register := 145, Value := 1);
	
	// Position Check variables
	bPosCheckNext : BOOL;
	nTaskType: INT := 1;
	bPosCheckAssignedUR3: BOOL;
	bPosCheckAssignedUR5: BOOL;
	bPosCheckCompleteUR3: BOOL;
	bPosCheckCompleteUR5: BOOL;
	nUR3PosCheckIndex : UINT := 1;
	nUR5PosCheckIndex : UINT := 1;
	
	bTestWait: BOOL;
END_VAR

(* =======================================================
Update veriables on every cycle
Multiple states are calculated on each cycle to aid in task assignment and tracking
======================================================= *)
// Update Task Status Information
fbUR3TaskStatusInfo(stTaskStatusInfo => stUR3TaskStatus);
fbUR5TaskStatusInfo(stTaskStatusInfo => stUR5TaskStatus);

// Triggers and Event Tracking
// Position Check Triggers
	IF Global.bEnablePosCheck THEN
		IF Global.bForcePosCheck OR Global.nPartsSincePosCheck >= Global.nPosCheckThreshold THEN
			bPosCheckNext := TRUE;
		END_IF
	END_IF
	// Reset Pos Check founter if it has been assigned for both robots
	IF bPosCheckCompleteUR3 AND bPosCheckCompleteUR5 THEN
		// if required trigger post check processing here
		Global.nPartsSincePosCheck := 0;
		bPosCheckAssignedUR3 := FALSE;
		bPosCheckAssignedUR5 := FALSE;
		bPosCheckCompleteUR3 := FALSE;
		bPosCheckCompleteUR5 := FALSE;
		bPosCheckNext := FALSE;
		Global.bForcePosCheck := FALSE;
	END_IF
// Stop Process Triggers
	StopAssignment_ftrig(CLK := Global.bActivateTaskAssignment);
	// Global interrupt
	// Interrupts
	IF StopAssignment_ftrig.Q THEN
		IF eUR3TaskState = E_RobotTaskStates.TaskSelection OR eUR3TaskState = E_RobotTaskStates.TaskTypeSelection THEN
			eUR3TaskState := E_RobotTaskStates.Idle;
		END_IF
		IF eUR5TaskState = E_RobotTaskStates.TaskSelection OR eUR5TaskState = E_RobotTaskStates.TaskTypeSelection THEN
			eUR5TaskState := E_RobotTaskStates.Idle;
		END_IF
	END_IF
//UR3 Task Triggers
	// Watch for UR3 task to be assigned
	UR3TaskActive_rtrig(CLK := stUR3TaskStatus.bInTask);
	// Watch for UR3 task to complete
	UR3TaskComplete_ftrig(CLK := stUR3TaskStatus.bInTask);
	// Watch for UR3 to start task action
	UR3ActionStart_rtrig(CLK := stUR3TaskStatus.bPerformingTaskAction);
	// Watch for UR3 to complete task action
	UR3ActionComplete_ftrig(CLK := stUR3TaskStatus.bPerformingTaskAction);
//UR5 Task Triggers
	// Watch for UR3 task to be assigned
	UR5TaskActive_rtrig(CLK := stUR5TaskStatus.bInTask);
	// Watch for UR3 task to complete
	UR5TaskComplete_ftrig(CLK := stUR5TaskStatus.bInTask);
	// Watch for UR3 to start task action
	UR5ActionStart_rtrig(CLK := stUR5TaskStatus.bPerformingTaskAction);
	// Watch for UR3 to complete task action
	UR5ActionComplete_ftrig(CLK := stUR5TaskStatus.bPerformingTaskAction);

// Calcualte part Time in Fixture
// Cycle through every workfixture
FOR nWorkFixtureIndex := 1 TO Global.nNumWorkFixtures DO
	// Calculate part times on every loop
	IF Global.arrWorkFixtures[nWorkFixtureIndex].stPart.bExists THEN
		Global.arrWorkFixtures[nWorkFixtureIndex].stPart.ntTimeInWorkfixture := 
			(Global.nCurrentTime - Global.arrWorkFixtures[nWorkFixtureIndex].stPart.ntInputPartPlaced)/10000000;
	ELSE
		Global.arrWorkFixtures[nWorkFixtureIndex].stPart.ntTimeInWorkfixture := 0;
	END_IF
END_FOR

// Update task type strings for visualization
IF eUR5TaskState = E_RobotTaskStates.TaskExecution THEN
	IF nUR5TargetTask = 1 THEN
		sUR5TargetTask := 'Input';
	ELSIF nUR5TargetTask = 2 THEN
		sUR5TargetTask := 'Output';
	END_IF
ELSE
	sUR5TargetTask := 'N/A';
END_IF


(* =======================================================
A state machine is used to handle the task state of the UR3 robot.
	Possible states include:
		- Idle - wait until process is in a mode to execute tasks
		- Task Type Selection - this is used to select between a drawing task or a measurement task. More can be added in the future
		- Task Selection - if no task is being executed, assesing if a task should be assigned
		- Task Assignment - packaging a task and transmititng it to the robot
		- Task Assignment Wait - waiting for task to be written to robot
		- Task Execution - waiting for robot to complete assigned task before going back to Idle
======================================================= *)
CASE eUR3TaskState OF
	E_RobotTaskStates.Idle: // Decides what to do based on system mode
		IF Global.bActivateTaskAssignment AND Global_Safety.UR3RedIND THEN
			eUR3TaskState := E_RobotTaskStates.TaskTypeSelection;
		END_IF
		// Reset Targets
		nUR3TargetWorkFixtureIndex := 0;
		nUR3TargetWorkframe := 0;
		nUR3TargetTask := 0;
		Global.bUR3InTask := FALSE;
	E_RobotTaskStates.TaskTypeSelection: // Should a position check test be performed
		IF bPosCheckNext AND NOT Global.bUR5InTask THEN
			IF NOT Global.bPosSensorReserved AND NOT bPosCheckCompleteUR3 THEN
				// Set Task Variables 
				nUR3TargetTask := 0; // 0 for Pos Check Program on robots
				Global.bPosSensorReserved := TRUE;
				bPosCheckAssignedUR3 := TRUE;
				nUR3PosCheckIndex := 1; // Index Value for Assignment of Sensor Inputs - Reset to 1
				eUR3TaskState := E_RobotTaskStates.TaskAssignment;
			END_IF
		ELSIF NOT bPosCheckNext THEN // else check if a different task that can be assigned
			// If a part exists and is not complete move to task selection
			IF Global.arrWorkFixtures[1].stPart.bExists AND NOT Global.arrWorkFixtures[1].stPart.bComplete THEN // If WF1 has a part that is not complete
				eUR3TaskState := E_RobotTaskStates.TaskSelection;
			ELSIF  Global.arrWorkFixtures[2].stPart.bExists AND NOT Global.arrWorkFixtures[2].stPart.bComplete THEN
				eUR3TaskState := E_RobotTaskStates.TaskSelection;
			END_IF
		END_IF
	E_RobotTaskStates.TaskSelection: // Monitoring and deciding if a task should be assigned
		// Reset MaxPartLagTime to help find longest lag time
		nMaxTimeInWF := 0;
		// Reset Targets
		nUR3TargetWorkFixtureIndex := 0;
		nUR3TargetWorkframe := 0;
		nUR3TargetTask := 0;
		// For each possible active workfixture
		FOR nWorkFixtureIndex := 1 TO Global.nNumWorkFixtures DO
			// If statement to identify if fixture/part can be worked on
			IF 	Global.arrWorkFixtures[nWorkFixtureIndex].stPart.bExists // part exists
			AND	NOT Global.arrWorkFixtures[nWorkFixtureIndex].stPart.bComplete // part not complete
			AND	NOT Global.arrWorkFixtures[nWorkFixtureIndex].bReserved THEN // fixture not reserved
				// Check to see if identified eligable part has been waiting the longest
				IF Global.arrWorkFixtures[nWorkFixtureIndex].stPart.ntTimeInWorkfixture > nMaxTimeInWF THEN
					// update max part lag time
					nMaxTimeInWF := Global.arrWorkFixtures[nWorkFixtureIndex].stPart.ntTimeInWorkfixture;
					// Record task, workframe and workfixture index
					nUR3TargetWorkframe := Global.arrWorkFixtures[nWorkFixtureIndex].nWorkframe;
					nUR3TargetPart := Global.arrWorkFixtures[nWorkFixtureIndex].stPart.nPartNumber;
					nUR3TargetWorkFixtureIndex := nWorkFixtureIndex;
					// if a viable target is found assign task
					eUR3TaskState := E_RobotTaskStates.TaskAssignment;
				END_IF
			END_IF
		END_FOR
		
		// Choose Task number 
		nUR3TargetTask := Global.nActiveUR3Task + 1; // 1 added for array indexing on radio button visu (starts at 0)
		(*
		FOR FUTURE VERSIONS - IF TASK IS TIED TO PART TYPE 
		Part type is stored in the following locaiton:
		Global.arrWorkFixtures[nUR3TargetWorkFixtureIndex].stPart.nPartType;
		*)
		
	E_RobotTaskStates.TaskAssignment: // Transmitting task to robot
		Global.bUR3InTask := TRUE;
		(* This section has two parts. 1) PLC handling and part tracking and 2) handling assignment to robot. *)
		// PLC Handling
		Global.arrWorkFixtures[nUR3TargetWorkFixtureIndex].bReserved := TRUE;
		
		// Robot Assignment Setup Handling
		fbWriteUR3Task.Task := nUR3TargetTask;
		fbWriteUR3Task.Workframe1 := nUR3TargetWorkframe;
		fbWriteUR3Task.PartNumber := nUR3TargetPart;
		fbWriteUR3Task.bExecute := TRUE;
		
		// Advance to waiting for assignment completion
		eUR3TaskState := E_RobotTaskStates.TaskAssignment_Wait;
	
	E_RobotTaskStates.TaskAssignment_Wait: 	// Waiting for task to be written
		IF NOT fbWriteUR3Task.bBusy THEN
			fbWriteUR3Task.bExecute :=FALSE;
			// record task assignment
			Global.arrWorkFixtures[nUR3TargetWorkFixtureIndex].stPart.ntTaskAssigned := Global.nCurrentTime;
			// change states
			eUR3TaskState := E_RobotTaskStates.TaskExecution;
		END_IF
			
	E_RobotTaskStates.TaskExecution: // Monitoring for completion of task
		// Recording Time at events
		IF UR3ActionStart_rtrig.Q THEN
			IF nUR3TargetTask = 0 THEN
				// record IO state here
				Global.UR3PosCheck[nUR3PosCheckIndex] := Global.bPosSensorState;
				nUR3PosCheckIndex := nUR3PosCheckIndex + 1;
				// tell robot to resume task
				fbUR3Resume.bExecute := TRUE;
			ELSE
				Global.arrWorkFixtures[nUR3TargetWorkFixtureIndex].stPart.ntTaskActionStart := Global.nCurrentTime;
			END_IF
		END_IF
		
		IF UR3ActionComplete_ftrig.Q THEN
			IF nUR3TargetTask = 0 THEN
				; // do noting
			ELSE
				Global.arrWorkFixtures[nUR3TargetWorkFixtureIndex].stPart.ntTaskActionComplete := Global.nCurrentTime;
			END_IF
		END_IF
		
		IF UR3TaskComplete_ftrig.Q THEN
			IF nUR3TargetTask = 0 THEN // If task completed was a pos check
				bPosCheckCompleteUR3 := TRUE;
				Global.bPosSensorReserved := FALSE;
				// (FOR UR integrated sensor) Global.UR3PosCheck := F_Word_To_16Bool(stUR3TaskStatus.nPosCheckValue);
			ELSE
				Global.arrWorkFixtures[nUR3TargetWorkFixtureIndex].stPart.bComplete := TRUE;
				Global.arrWorkFixtures[nUR3TargetWorkFixtureIndex].bReserved := FALSE;
				// Record Complete
				Global.arrWorkFixtures[nUR3TargetWorkFixtureIndex].stPart.ntTaskComplete := Global.nCurrentTime;
			END_IF
			// Go back to idle state
			eUR3TaskState := E_RobotTaskStates.Idle;
		END_IF
END_CASE

(* =======================================================
UR5
A state machine is used to handle the task state of the UR5 robot.
	Possible states include:
		- Idle - wait until process is in a mode to execute tasks
		- Task Selection - if no task is being executed, assesing if a task should be assigned
		- Task Assignment - packaging a task and transmititng it to the robot
		- Task Assignment Wait - waiting for task to be written to robot
		- Task Execution - waiting for robot to complete assigned task before going back to Idle
======================================================= *)
CASE eUR5TaskState OF
	E_RobotTaskStates.Idle: // Decides what to do based on system mode
		IF Global.bActivateTaskAssignment AND Global_Safety.UR5RedIND THEN
			eUR5TaskState := E_RobotTaskStates.TaskTypeSelection;
		END_IF
		// Reset Targets
		nUR5TargetWorkFixtureIndex := 0;
		nUR5TargetInputFixtureIndex := 0;
		nUR5TargetOutputFixtureIndex := 0;
		nUR5TargetPickFrame := 0;
		nUR5TargetPlaceFrame := 0;
		nUR5TargetTask := 0;
		nMaxTimeInWF := 0;
		Global.bUR5InTask := FALSE;
	E_RobotTaskStates.TaskTypeSelection: // Should a position check test be performed
		IF bPosCheckNext AND NOT Global.bUR3InTask THEN
			// Choose Task number 
			IF NOT Global.bPosSensorReserved AND NOT bPosCheckCompleteUR5 THEN
				nUR5TargetTask := 0; // 0 for Pos Check Program on robots
				Global.bPosSensorReserved := TRUE;
				bPosCheckAssignedUR5 := TRUE;
				nUR5PosCheckIndex := 1; // Index Value for Assignment of Sensor Inputs - Reset to 1
				eUR5TaskState := E_RobotTaskStates.TaskAssignment;
			END_IF
		ELSIF NOT bPosCheckNext THEN  
			// else it is a different task that must be assigned
			// If an input part exists or a complete part exists
			IF Global.arrInputFixtures[1].stPart.bExists OR Global.arrWorkFixtures[1].stPart.bComplete OR Global.arrWorkFixtures[2].stPart.bComplete THEN 
				eUR5TaskState := E_RobotTaskStates.TaskSelection;
			END_IF
		END_IF
	E_RobotTaskStates.TaskSelection: // Monitoring and deciding if a task should be assigned
		// OUTPUT - Find possible part OUTPUTS
		nUR5TargetPickFrame := 0;
		nUR5TargetPlaceFrame := 0;
		// For each possible active workfixture
		FOR nWorkFixtureIndex := 1 TO Global.nNumWorkFixtures DO
			IF Global.arrWorkFixtures[nWorkFixtureIndex].stPart.bExists // part exists
			AND Global.arrWorkFixtures[nWorkFixtureIndex].stPart.bComplete // part is complete (ready for output)
			AND NOT Global.arrWorkFixtures[nWorkFixtureIndex].bReserved THEN // fixture is not reserved
				// Determine if it has been waiting the longest (FIFO)
				IF Global.arrWorkFixtures[nWorkFixtureIndex].stPart.ntTimeInWorkfixture > nMaxTimeInWF THEN
					// update max part lag time
					nMaxTimeInWF := Global.arrWorkFixtures[nWorkFixtureIndex].stPart.ntTimeInWorkfixture;
					// Record task, workframe and workfixture index
					nUR5TargetWorkFixtureIndex := nWorkFixtureIndex;
					nUR5TargetPart := Global.arrWorkFixtures[nWorkFixtureIndex].stPart.nPartNumber;
					nUR5TargetPickFrame := Global.arrWorkFixtures[nWorkFixtureIndex].nWorkframe;
				END_IF
			END_IF
		END_FOR
		// For each possible output fixture
		FOR nOutputFixtureIndex := 1 TO Global.nNumOutputFixtures DO
			// find first available input part (in order, NO FIFO)
			IF NOT Global.arrOutputFixtures[nOutputFixtureIndex].stPart.bExists THEN
				// Record target information
				nUR5TargetOutputFixtureIndex := nOutputFixtureIndex;
				nUR5TargetPlaceFrame := Global.arrOutputFixtures[nOutputFixtureIndex].nWorkframe;
				// if a viable target is found assign task
			END_IF
			IF nUR5TargetPlaceFrame > 0 THEN
					// exit for loop
					EXIT;
			END_IF
		END_FOR
		// assign task type if a task was found
		IF nUR5TargetPickFrame <> 0 AND nUR5TargetPlaceFrame <> 0 THEN // pick and place found
			nUR5TargetTask := 2; // 2 for output task
			eUR5TaskState := E_RobotTaskStates.TaskAssignment;
		END_IF
		// INPUT - If output is not assigned find possible INPUTS
		
		IF nUR5TargetTask <> 2 THEN
			nUR5TargetPickFrame := 0;
			nUR5TargetPlaceFrame := 0;
			// check if each work fixture is empty
			FOR nWorkFixtureIndex := 1 TO Global.nNumWorkFixtures DO
				IF NOT Global.arrWorkFixtures[nWorkFixtureIndex].stPart.bExists // no part in fixture
				AND NOT Global.arrWorkFixtures[nWorkFixtureIndex].bReserved THEN // fixture is not reserved
					// record target informaiton
					nUR5TargetWorkFixtureIndex := nWorkFixtureIndex;
					nUR5TargetPlaceFrame := Global.arrWorkFixtures[nWorkFixtureIndex].nWorkframe;
				END_IF
				IF nUR5TargetPlaceFrame > 0 THEN
					// exit for loop
					EXIT;
				END_IF
			END_FOR
			// check for available part in input
			FOR nInputFixtureIndex := 1 TO Global.nNumInputFixtures DO
				// find first available input part (in order, NO FIFO)
				IF 	Global.arrInputFixtures[nInputFixtureIndex].stPart.bExists THEN
					// Record target information
					nUR5TargetInputFixtureIndex := nInputFixtureIndex;
					nUR5TargetPart := Global.arrInputFixtures[nInputFixtureIndex].stPart.nPartNumber;
					nUR5TargetPickFrame := Global.arrInputFixtures[nInputFixtureIndex].nWorkframe;
				END_IF
				IF nUR5TargetPickFrame > 0 THEN
					// exit for loop
					EXIT;
				END_IF
			END_FOR
			// check if task was assigned
			IF nUR5TargetPickFrame <> 0 AND nUR5TargetPlaceFrame <> 0 THEN
				nUR5TargetTask := 1; // 1 for input task
				eUR5TaskState := E_RobotTaskStates.TaskAssignment;
			END_IF
		END_IF
	E_RobotTaskStates.TaskAssignment: // Transmitting task to robot
		(* This section has two parts. 1) handling PLC tracking side and 2) handling assignment to robot. *)
		// PLC Handling
		Global.bUR5InTask  := TRUE;
		IF nUR5TargetTask = 1 THEN // If input task
			Global.arrInputFixtures[nUR5TargetInputFixtureIndex].bReserved := TRUE;
			// Record task information
			Global.arrInputFixtures[nUR5TargetInputFixtureIndex].stPart.nInputPosition := nUR5TargetPickFrame;
			Global.arrInputFixtures[nUR5TargetInputFixtureIndex].stPart.nWorkFixture := nUR5TargetPlaceFrame;
		ELSIF nUR5TargetTask = 2 THEN // If output task
			Global.arrOutputFixtures[nUR5TargetOutputFixtureIndex].bReserved := TRUE;
			// Record task information
			Global.arrWorkFixtures[nUR5TargetWorkFixtureIndex].stPart.nOutputPosition := nUR5TargetPlaceFrame;
		END_IF
		
		Global.arrWorkFixtures[nUR5TargetWorkFixtureIndex].bReserved := TRUE;
		
		
		// Robot Assignment Setup Handling
		fbWriteUR5Task.Task := nUR5TargetTask;
		fbWriteUR5Task.Workframe1 := nUR5TargetPickFrame;
		fbWriteUR5Task.Workframe2 := nUR5TargetPlaceFrame;
		fbWriteUR5Task.PartNumber := nUR5TargetPart;
		fbWriteUR5Task.bExecute := TRUE;
		
		// Advance to waiting for assignment completion
		eUR5TaskState := E_RobotTaskStates.TaskAssignment_Wait;
	
	E_RobotTaskStates.TaskAssignment_Wait: 	// Waiting for task to be written
		IF NOT fbWriteUR5Task.bBusy THEN
			fbWriteUR5Task.bExecute :=FALSE;
			// record assignment time
			IF nUR5TargetTask = 1 THEN // If input task
				Global.arrInputFixtures[nUR5TargetInputFixtureIndex].stPart.ntPickFromInputAssigned := Global.nCurrentTime;
			ELSIF nUR5TargetTask = 2 THEN // If output task
				Global.arrWorkFixtures[nUR5TargetWorkFixtureIndex].stPart.ntPickFromWFAssigned := Global.nCurrentTime;
			END_IF
			
			// change states
			eUR5TaskState := E_RobotTaskStates.TaskExecution;
		END_IF
			
	E_RobotTaskStates.TaskExecution: // Monitoring for completion of task
		// Handle task events
		IF UR5ActionStart_rtrig.Q THEN // when action starts
			IF nUR5TargetTask = 0 THEN
				// record IO state here
				Global.UR5PosCheck[nUR5PosCheckIndex] := Global.bPosSensorState;
				nUR5PosCheckIndex := nUR5PosCheckIndex + 1;
				// tell robot to resume task
				fbUR5Resume.bExecute := TRUE;
			// record Action start time and handle part movement
			ELSIF nUR5TargetTask = 1 THEN // If input task
				Global.arrInputFixtures[nUR5TargetInputFixtureIndex].stPart.ntInputPartPicked := Global.nCurrentTime;
				Global.stPartInTransit := Global.arrInputFixtures[nUR5TargetInputFixtureIndex].stPart;
				Global.arrInputFixtures[nUR5TargetInputFixtureIndex].stPart := Global.stNullPart;
			ELSIF nUR5TargetTask = 2 THEN // If output task
				Global.arrWorkFixtures[nUR5TargetWorkFixtureIndex].stPart.ntOutputPartPicked := Global.nCurrentTime;
				Global.stPartInTransit := Global.arrWorkFixtures[nUR5TargetWorkFixtureIndex].stPart;
				Global.arrWorkFixtures[nUR5TargetWorkFixtureIndex].stPart := Global.stNullPart;
			END_IF
		END_IF
		IF UR5ActionComplete_ftrig.Q THEN
			IF nUR5TargetTask = 0 THEN
				; // do noting
			// record Action Complete time and handle part movement
			ELSIF nUR5TargetTask = 1 THEN // If input task
				Global.arrWorkFixtures[nUR5TargetWorkFixtureIndex].stPart := Global.stPartInTransit;
				Global.arrWorkFixtures[nUR5TargetWorkFixtureIndex].stPart.ntInputPartPlaced := Global.nCurrentTime;
				Global.stPartInTransit := Global.stNullPart;
			ELSIF nUR5TargetTask = 2 THEN // If output task
				Global.arrOutputFixtures[nUR5TargetOutputFixtureIndex].stPart := Global.stPartInTransit;
				Global.arrOutputFixtures[nUR5TargetOutputFixtureIndex].stPart.ntOutputPartPlaced := Global.nCurrentTime;
				Global.stPartInTransit := Global.stNullPart;
			END_IF
		END_IF
		
		IF UR5TaskComplete_ftrig.Q THEN
			// record Action Complete time and handle part movement
			IF nUR5TargetTask = 0 THEN // If task completed was a pos check
				bPosCheckCompleteUR5 := TRUE;
				Global.bPosSensorReserved := FALSE;
				// Global.UR5PosCheck := F_Word_To_16Bool(stUR5TaskStatus.nPosCheckValue);
			ELSIF nUR5TargetTask = 1 THEN // If input task
				Global.arrWorkFixtures[nUR5TargetWorkFixtureIndex].stPart.ntPlaceInWFComplete := Global.nCurrentTime;
				Global.arrWorkFixtures[nUR5TargetWorkFixtureIndex].bReserved := FALSE;
				Global.arrInputFixtures[nUR5TargetInputFixtureIndex].bReserved := FALSE;
			ELSIF nUR5TargetTask = 2 THEN // If output task
				Global.arrOutputFixtures[nUR5TargetOutputFixtureIndex].stPart.ntPlaceInOutputComplete := Global.nCurrentTime;
				Global.arrOutputFixtures[nUR5TargetOutputFixtureIndex].bReserved := FALSE;
				Global.arrWorkFixtures[nUR5TargetWorkFixtureIndex].bReserved := FALSE;
				// Pos Check Part Counting
				Global.nPartsSincePosCheck := Global.nPartsSincePosCheck + 1;
			END_IF
			// Go back to idle state
			eUR5TaskState := E_RobotTaskStates.Idle;
		END_IF
END_CASE

(* =======================================================
Function block Calls
======================================================= *)
fbWriteUR3Task();
fbWriteUR5Task();
fbUR3Resume();
fbUR5Resume();

END_PROGRAM

// ---- POUs/Modbus POUs/FB_mbReadRobotTaskStatusInfo.TcPOU
FUNCTION_BLOCK FB_mbReadRobotTaskStatusInfo
VAR_INPUT
	Robot : STRING;
END_VAR
VAR_OUTPUT
	stTaskStatusInfo : ST_RobotTaskStatusInfo;
END_VAR
VAR
	Value : ARRAY [1..12] OF WORD;
	mbRead : FB_mbReadRegs;
	state : int;
END_VAR

(* 
FB_mbReadRobotStatusInfo - Function Block that can be called to read a Robot status registers: 128-139
	INPUTS:
		- Robot : Sting, 'UR5' or 'UR3'
	OUTPUTS
		- RobotTaskStatus : WORD;
		- ZoneOccupied : WORD;
		- IsInTask : BOOL;
		- IsPerformingTaskAction : BOOL;
*)

// Set function block vairables
mbRead.nQuantity := 12;
mbRead.cbLength := 24;

IF Robot='UR5' THEN
	mbRead.sIPAddr := Global.stUR5.IP;
	mbRead.nTCPPort := Global.stUR5.mbPort;
	mbRead.nUnitID := Global.stUR5.unitID;
ELSIF Robot='UR3' THEN
	mbRead.sIPAddr := Global.stUR3.IP;
	mbRead.nTCPPort := Global.stUR3.mbPort;
	mbRead.nUnitID := Global.stUR3.unitID;
END_IF

mbRead.pDestAddr := ADR(Value);
mbRead.nMBAddr := 128;

// Set/Determine State of Function block
CASE state OF
	0:
		mbRead.bExecute := TRUE;
		state := 10;
	10:
		IF NOT mbRead.bBusy THEN
			mbRead.bExecute :=FALSE;
			state := 20;
		END_IF
	20:
		stTaskStatusInfo.nRobotTaskStatus := Value[1];
		stTaskStatusInfo.nZoneOccupied := Value[2];
		stTaskStatusInfo.bInTask := INT_TO_BOOL(Value[3]);
		stTaskStatusInfo.bPerformingTaskAction := INT_TO_BOOL(Value[4]);
		
		IF stTaskStatusInfo.nRobotTaskStatus = 1 THEN
			stTaskStatusInfo.sRobotStatus := 'Waiting for Task Assignment';
		ELSIF stTaskStatusInfo.nRobotTaskStatus = 2 THEN
			stTaskStatusInfo.sRobotStatus := 'Executing Assigned Task';
		END_IF

		state := 0;
END_CASE

// Run function block
mbRead();

END_FUNCTION_BLOCK

// ---- POUs/Modbus POUs/FB_mbWriteRobotTask.TcPOU
FUNCTION_BLOCK FB_mbWriteRobotTask
VAR_INPUT
	bExecute : BOOL;
	Robot : STRING;
	// Keep task and workframe together for memory allocation
	Task : WORD;
	Workframe1 : WORD;
	Workframe2 : WORD;
	PartNumber : WORD;
	ResumeTask : WORD;
END_VAR
VAR_OUTPUT
	bBusy : BOOL;
END_VAR
VAR
	message : ARRAY [1..13] OF WORD;
	mbWrite : FB_mbWriteRegs;
	state : INT;
	NewTask : WORD;
END_VAR

(* 
FB_mbWriteRobotTask - Function Block that can be called to write robot
Registers 140-149
	See IO_Documentation.xlsx file for register mapping summary
		
*)
IF bExecute THEN
	// Set/Determine State of Function block
	CASE state OF
		0:
			(* Build Message to send *)
			// Newtask always equals 1 when sending a new task
			NewTask := 1;
			ResumeTask := 0;
			// put variable being transfered into organized memory space
			message[1] := NewTask;
			message[2] := Task;
			message[3] := Workframe1;
			message[4] := Workframe2;
			message[5] := PartNumber;
			message[6] := ResumeTask;
			
			(* Set function block vairables *)
			// package size information
			mbWrite.nQuantity := 13;
			mbWrite.cbLength := 26;
			
			// Robot specific information
			IF Robot='UR5' THEN
				mbWrite.sIPAddr := Global.stUR5.IP;
				mbWrite.nTCPPort := Global.stUR5.mbPort;
				mbWrite.nUnitID := Global.stUR5.unitID;
				
				message[7] := Global.stUR5.InducedJErrorType;
				message[8] := Global.stUR5.InducedJointError[1];
				message[9] := Global.stUR5.InducedJointError[2];
				message[10] := Global.stUR5.InducedJointError[3];
				message[11] := Global.stUR5.InducedJointError[4];
				message[12] := Global.stUR5.InducedJointError[5];
				message[13] := Global.stUR5.InducedJointError[6];
			ELSIF Robot='UR3' THEN
				mbWrite.sIPAddr := Global.stUR3.IP;
				mbWrite.nTCPPort := Global.stUR3.mbPort;
				mbWrite.nUnitID := Global.stUR3.unitID;
				
				message[7] := Global.stUR3.InducedJErrorType;
				message[8] := Global.stUR3.InducedJointError[1];
				message[9] := Global.stUR3.InducedJointError[2];
				message[10] := Global.stUR3.InducedJointError[3];
				message[11] := Global.stUR3.InducedJointError[4];
				message[12] := Global.stUR3.InducedJointError[5];
				message[13] := Global.stUR3.InducedJointError[6];
			END_IF
			
			// source and destination information
			mbWrite.pSrcAddr := ADR(message);
			mbWrite.nMBAddr := 140;
			
			// Execute MODBUS Write
			mbWrite.bExecute := TRUE;
			
			// Set fuctionblock busy bit
			bBusy := TRUE;
			
			// Advance to waiting for completion state
			state := 10;
		10:
			IF NOT mbWrite.bBusy THEN
				mbWrite.bExecute :=FALSE;
				bBusy := FALSE;
				state := 0;
			END_IF
	END_CASE
	
	// Run function block
	mbWrite();

END_IF

END_FUNCTION_BLOCK

// ---- POUs/Modbus POUs/FB_mbWriteSingleReg.TcPOU
FUNCTION_BLOCK FB_mbWriteSingleReg
VAR_INPUT
	bExecute : BOOL;
	Robot : STRING;
	Register : WORD;
	Value : WORD;
END_VAR
VAR_OUTPUT
	bBusy : BOOL;
END_VAR
VAR
	mbWrite : FB_mbWriteRegs;
	state : int;
END_VAR

(* 
FB_mbWriteSingleReg - Function Block that can be called to write a single MODBUS register
	INPUTS:
		- Robot: 'UR5' or 'UR3'
		- Register: register number to write
		- Value: value to write
	OUTPUTS
		
*)

IF bExecute THEN
	// Set/Determine State of Function block
	CASE state OF
		0:
			// Set function block vairables
			mbWrite.nQuantity := 1;
			mbWrite.cbLength := 2;
			
			IF Robot='UR5' THEN
				mbWrite.sIPAddr := Global.stUR5.IP;
				mbWrite.nTCPPort := Global.stUR5.mbPort;
				mbWrite.nUnitID := Global.stUR5.unitID;
			ELSIF Robot='UR3' THEN
				mbWrite.sIPAddr := Global.stUR3.IP;
				mbWrite.nTCPPort := Global.stUR3.mbPort;
				mbWrite.nUnitID := Global.stUR3.unitID;
			END_IF
			
			mbWrite.pSrcAddr := ADR(Value);
			mbWrite.nMBAddr := Register;
			mbWrite.bExecute := TRUE;
			
			// Set fuctionblock busy bit
			bBusy := TRUE;
			
			state := 10;
	
		10:
			IF NOT mbWrite.bBusy THEN
				mbWrite.bExecute :=FALSE;
				state := 0;
			END_IF
	END_CASE
	
	// Run function block
	mbWrite();
END_IF

END_FUNCTION_BLOCK

// ---- POUs/F_Word_To_16Bool.TcPOU
FUNCTION F_Word_To_16Bool : ST_16Bool
VAR_INPUT
	value : WORD;
END_VAR
VAR
END_VAR

F_Word_To_16Bool.var1 := INT_TO_BOOL(2#0000_0000_0000_0001 AND value);
F_Word_To_16Bool.var2 := INT_TO_BOOL(2#0000_0000_0000_0010 AND value);
F_Word_To_16Bool.var3 := INT_TO_BOOL(2#0000_0000_0000_0100 AND value);
F_Word_To_16Bool.var4 := INT_TO_BOOL(2#0000_0000_0000_1000 AND value);
F_Word_To_16Bool.var5 := INT_TO_BOOL(2#0000_0000_0001_0000 AND value);
F_Word_To_16Bool.var6 := INT_TO_BOOL(2#0000_0000_0010_0000 AND value);
F_Word_To_16Bool.var7 := INT_TO_BOOL(2#0000_0000_0100_0000 AND value);
F_Word_To_16Bool.var8 := INT_TO_BOOL(2#0000_0000_1000_0000 AND value);
F_Word_To_16Bool.var9 := INT_TO_BOOL(2#0000_0001_0000_0000 AND value);
F_Word_To_16Bool.var10 := INT_TO_BOOL(2#0000_0010_0000_0000 AND value);
F_Word_To_16Bool.var11 := INT_TO_BOOL(2#0000_0100_0000_0000 AND value);
F_Word_To_16Bool.var12 := INT_TO_BOOL(2#0000_1000_0000_0000 AND value);
F_Word_To_16Bool.var13 := INT_TO_BOOL(2#0001_0000_0000_0000 AND value);
F_Word_To_16Bool.var14 := INT_TO_BOOL(2#0010_0000_0000_0000 AND value);
F_Word_To_16Bool.var15 := INT_TO_BOOL(2#0100_0000_0000_0000 AND value);
F_Word_To_16Bool.var16 := INT_TO_BOOL(2#1000_0000_0000_0000 AND value);

END_FUNCTION

// ---- POUs/P_InitializeSystem.TcPOU
PROGRAM P_InitializeSystem
VAR
END_VAR

END_PROGRAM

